LIN {X 0,Y 512.097,Z 685.03,A -85,B 0,C 180,E1 4897.992,E2 4897.992} C_VEL
LIN {X 0,Y 512.114,Z 685.03,A -85,B 0,C 180,E1 4902.666,E2 4902.666} C_VEL
LIN {X 0,Y 512.18,Z 685.03,A -85,B 0,C 180,E1 4907.439,E2 4907.439} C_VEL
LIN {X 0,Y 512.504,Z 685.03,A -85,B 0,C 180,E1 4913.923,E2 4913.923} C_VEL
LIN {X 0,Y 527.673,Z 717.271,A -85,B 0,C 180,E1 4915.573,E2 4915.573} C_VEL
LIN {X 0,Y 526.848,Z 777.404,A -85,B 0,C 180,E1 4916.651,E2 4916.651} C_VEL
LIN {X 0,Y 525.113,Z 815.762,A -85,B 0,C 180,E1 4917.972,E2 4917.972} C_VEL
LIN {X 0,Y 522.678,Z 854.116,A -85,B 0,C 180,E1 4920.009,E2 4920.009} C_VEL
LIN {X 0,Y 520.002,Z 889.911,A -85,B 0,C 180,E1 4922.686,E2 4922.686} C_VEL
LIN {X 0,Y 517.704,Z 920.346,A -85,B 0,C 180,E1 4925.724,E2 4925.724} C_VEL
LIN {X 0,Y 515.761,Z 947.251,A -85,B 0,C 180,E1 4929.222,E2 4929.222} C_VEL
LIN {X 0,Y 514.265,Z 970.27,A -85,B 0,C 180,E1 4933.156,E2 4933.156} C_VEL
LIN {X 0,Y 513.451,Z 987.984,A -85,B 0,C 180,E1 4937.266,E2 4937.266} C_VEL
LIN {X 0,Y 513.157,Z 1000.678,A -85,B 0,C 180,E1 4941.545,E2 4941.545} C_VEL
LIN {X 0,Y 512.98,Z 1006.957,A -85,B 0,C 180,E1 4944.937,E2 4944.937} C_VEL
LIN {X 0,Y 513,Z 1010.088,A -85,B 0,C 180,E1 4948.314,E2 4948.314} C_VEL
LIN {X 0,Y 513.108,Z 1010.088,A -85,B 0,C 180,E1 4951.685,E2 4951.685} C_VEL
LIN {X 0,Y 513.105,Z 1005.755,A -85,B 0,C 180,E1 4955.908,E2 4955.908} C_VEL
LIN {X 0,Y 513.209,Z 996.305,A -85,B 0,C 180,E1 4960.161,E2 4960.161} C_VEL
LIN {X 0,Y 513.736,Z 982.178,A -85,B 0,C 180,E1 4964.236,E2 4964.236} C_VEL
LIN {X 0,Y 514.8,Z 962.363,A -85,B 0,C 180,E1 4968.326,E2 4968.326} C_VEL
LIN {X 0,Y 516.536,Z 936.319,A -85,B 0,C 180,E1 4972.32,E2 4972.32} C_VEL
LIN {X 0,Y 518.821,Z 905.459,A -85,B 0,C 180,E1 4975.866,E2 4975.866} C_VEL
LIN {X 0,Y 521.366,Z 871.94,A -85,B 0,C 180,E1 4978.762,E2 4978.762} C_VEL
LIN {X 0,Y 523.841,Z 836.554,A -85,B 0,C 180,E1 4981.017,E2 4981.017} C_VEL
LIN {X 0,Y 525.931,Z 799.056,A -85,B 0,C 180,E1 4982.681,E2 4982.681} C_VEL
LIN {X 0,Y 527.45,Z 761.276,A -85,B 0,C 180,E1 4983.702,E2 4983.702} C_VEL
LIN {X 0,Y 527.348,Z 716.349,A -85,B 0,C 180,E1 4984.466,E2 4984.466} C_VEL
LIN {X 0,Y 512.508,Z 685.03,A -85,B 0,C 180,E1 4986.077,E2 4986.077} C_VEL
LIN {X 0,Y 512.162,Z 685.03,A -85,B 0,C 180,E1 4992.66,E2 4992.66} C_VEL
LIN {X 0,Y 512.266,Z 685.03,A -85,B 0,C 180,E1 4999.604,E2 4999.604} C_VEL
LIN {X 0,Y 512.378,Z 685.03,A -85,B 0,C 180,E1 5005.55,E2 5005.55} C_VEL
LIN {X 0,Y 512.303,Z 685.03,A -85,B 0,C 180,E1 5009.95,E2 5009.95} C_VEL
LIN {X 0,Y 512.329,Z 685.03,A -85,B 0,C 180,E1 5015.932,E2 5015.932} C_VEL
LIN {X 0,Y 512.467,Z 685.03,A -85,B 0,C 180,E1 5021.099,E2 5021.099} C_VEL
LIN {X 0,Y 512.624,Z 685.03,A -85,B 0,C 180,E1 5026.377,E2 5026.377} C_VEL
LIN {X 0,Y 512.65,Z 685.03,A -85,B 0,C 180,E1 5031.534,E2 5031.534} C_VEL
LIN {X 0,Y 512.92,Z 685.03,A -85,B 0,C 180,E1 5036.624,E2 5036.624} C_VEL
LIN {X 0,Y 513.012,Z 685.03,A -85,B 0,C 180,E1 5041.682,E2 5041.682} C_VEL
LIN {X 0,Y 512.789,Z 685.03,A -85,B 0,C 180,E1 5046.756,E2 5046.756} C_VEL
LIN {X 0,Y 512.606,Z 685.03,A -85,B 0,C 180,E1 5051.888,E2 5051.888} C_VEL
LIN {X 0,Y 512.525,Z 685.03,A -85,B 0,C 180,E1 5057.118,E2 5057.118} C_VEL
LIN {X 0,Y 512.414,Z 685.03,A -85,B 0,C 180,E1 5062.504,E2 5062.504} C_VEL
LIN {X 0,Y 512.263,Z 685.03,A -85,B 0,C 180,E1 5068.114,E2 5068.114} C_VEL
LIN {X 0,Y 512.159,Z 685.03,A -85,B 0,C 180,E1 5074.414,E2 5074.414} C_VEL
LIN {X 0,Y 512.28,Z 685.03,A -85,B 0,C 180,E1 5080.386,E2 5080.386} C_VEL
LIN {X 0,Y 512.179,Z 685.03,A -85,B 0,C 180,E1 5085.001,E2 5085.001} C_VEL
LIN {X 0,Y 512.172,Z 685.03,A -85,B 0,C 180,E1 5091.778,E2 5091.778} C_VEL
LIN {X 0,Y 512.431,Z 685.03,A -85,B 0,C 180,E1 5097.991,E2 5097.991} C_VEL
LIN {X 0,Y 512.52,Z 685.291,A -85,B 0,C 180,E1 5101.148,E2 5101.148} C_VEL
LIN {X 0,Y 521.072,Z 714.374,A -85,B 0,C 180,E1 5103.391,E2 5103.391} C_VEL
LIN {X 0,Y 518.767,Z 750.096,A -85,B 0,C 180,E1 5105.855,E2 5105.855} C_VEL
LIN {X 0,Y 516.704,Z 780.667,A -85,B 0,C 180,E1 5108.764,E2 5108.764} C_VEL
LIN {X 0,Y 515.025,Z 806.913,A -85,B 0,C 180,E1 5112.149,E2 5112.149} C_VEL
LIN {X 0,Y 513.952,Z 827.068,A -85,B 0,C 180,E1 5115.644,E2 5115.644} C_VEL
LIN {X 0,Y 513.394,Z 843.521,A -85,B 0,C 180,E1 5119.617,E2 5119.617} C_VEL
LIN {X 0,Y 513.147,Z 853.42,A -85,B 0,C 180,E1 5123.245,E2 5123.245} C_VEL
LIN {X 0,Y 513.102,Z 858.723,A -85,B 0,C 180,E1 5126.628,E2 5126.628} C_VEL
LIN {X 0,Y 513.002,Z 860.423,A -85,B 0,C 180,E1 5130.379,E2 5130.379} C_VEL
LIN {X 0,Y 513.086,Z 857.628,A -85,B 0,C 180,E1 5134.216,E2 5134.216} C_VEL
LIN {X 0,Y 513.282,Z 849.065,A -85,B 0,C 180,E1 5138.453,E2 5138.453} C_VEL
LIN {X 0,Y 513.64,Z 835.976,A -85,B 0,C 180,E1 5142.298,E2 5142.298} C_VEL
LIN {X 0,Y 514.466,Z 816.847,A -85,B 0,C 180,E1 5146.179,E2 5146.179} C_VEL
LIN {X 0,Y 515.912,Z 793.18,A -85,B 0,C 180,E1 5149.655,E2 5149.655} C_VEL
LIN {X 0,Y 517.757,Z 765.125,A -85,B 0,C 180,E1 5152.734,E2 5152.734} C_VEL
LIN {X 0,Y 519.902,Z 732.834,A -85,B 0,C 180,E1 5155.348,E2 5155.348} C_VEL
LIN {X 0,Y 520.429,Z 711.081,A -85,B 0,C 180,E1 5156.776,E2 5156.776} C_VEL
LIN {X 0,Y 513.339,Z 688.629,A -85,B 0,C 180,E1 5158.542,E2 5158.542} C_VEL
LIN {X 0,Y 512.428,Z 685.03,A -85,B 0,C 180,E1 5158.781,E2 5158.781} C_VEL
LIN {X 0,Y 512.245,Z 685.03,A -85,B 0,C 180,E1 5164.44,E2 5164.44} C_VEL
LIN {X 0,Y 512.172,Z 685.03,A -85,B 0,C 180,E1 5170.404,E2 5170.404} C_VEL
LIN {X 0,Y 512.18,Z 685.03,A -85,B 0,C 180,E1 5175.01,E2 5175.01} C_VEL
LIN {X 0,Y 512.298,Z 685.03,A -85,B 0,C 180,E1 5179.982,E2 5179.982} C_VEL
LIN {X 0,Y 512.199,Z 685.03,A -85,B 0,C 180,E1 5185.968,E2 5185.968} C_VEL
LIN {X 0,Y 512.303,Z 685.03,A -85,B 0,C 180,E1 5192.086,E2 5192.086} C_VEL
LIN {X 0,Y 512.422,Z 685.03,A -85,B 0,C 180,E1 5197.496,E2 5197.496} C_VEL
LIN {X 0,Y 512.61,Z 685.03,A -85,B 0,C 180,E1 5202.885,E2 5202.885} C_VEL
LIN {X 0,Y 512.652,Z 685.03,A -85,B 0,C 180,E1 5208.113,E2 5208.113} C_VEL
LIN {X 0,Y 512.68,Z 685.03,A -85,B 0,C 180,E1 5213.242,E2 5213.242} C_VEL
LIN {X 0,Y 512.709,Z 685.03,A -85,B 0,C 180,E1 5218.317,E2 5218.317} C_VEL
LIN {X 0,Y 512.758,Z 685.03,A -85,B 0,C 180,E1 5223.377,E2 5223.377} C_VEL
LIN {X 0,Y 512.593,Z 685.03,A -85,B 0,C 180,E1 5228.467,E2 5228.467} C_VEL
LIN {X 0,Y 512.526,Z 685.03,A -85,B 0,C 180,E1 5233.689,E2 5233.689} C_VEL
LIN {X 0,Y 512.406,Z 685.03,A -85,B 0,C 180,E1 5239.546,E2 5239.546} C_VEL
LIN {X 0,Y 512.335,Z 685.03,A -85,B 0,C 180,E1 5244.354,E2 5244.354} C_VEL
LIN {X 0,Y 512.197,Z 685.03,A -85,B 0,C 180,E1 5250.057,E2 5250.057} C_VEL
LIN {X 0,Y 512.084,Z 685.03,A -85,B 0,C 180,E1 5256.112,E2 5256.112} C_VEL
LIN {X 0,Y 512.097,Z 685.03,A -85,B 0,C 180,E1 5257.992,E2 5257.992} C_VEL
LIN {X 0,Y 509.625,Z 685.03,A -85,B 0,C 180,E1 5259.422,E2 5259.422} C_VEL
LIN {X 0,Y 504.094,Z 685.03,A -85,B 0,C 180,E1 5261.814,E2 5261.814} C_VEL
LIN {X 0,Y 504.227,Z 685.03,A -85,B 0,C 180,E1 5268.432,E2 5268.432} C_VEL
LIN {X 0,Y 504.534,Z 685.03,A -85,B 0,C 180,E1 5273.399,E2 5273.399} C_VEL
LIN {X 0,Y 515.554,Z 708.405,A -85,B 0,C 180,E1 5274.539,E2 5274.539} C_VEL
LIN {X 0,Y 521.274,Z 720.033,A -85,B 0,C 180,E1 5275.135,E2 5275.135} C_VEL
LIN {X 0,Y 520.263,Z 777.402,A -85,B 0,C 180,E1 5276.172,E2 5276.172} C_VEL
LIN {X 0,Y 518.336,Z 816.284,A -85,B 0,C 180,E1 5277.529,E2 5277.529} C_VEL
LIN {X 0,Y 515.69,Z 854.113,A -85,B 0,C 180,E1 5279.56,E2 5279.56} C_VEL
LIN {X 0,Y 512.844,Z 889.613,A -85,B 0,C 180,E1 5282.245,E2 5282.245} C_VEL
LIN {X 0,Y 510.294,Z 920.539,A -85,B 0,C 180,E1 5285.372,E2 5285.372} C_VEL
LIN {X 0,Y 508.137,Z 947.251,A -85,B 0,C 180,E1 5288.895,E2 5288.895} C_VEL
LIN {X 0,Y 506.553,Z 970.269,A -85,B 0,C 180,E1 5292.892,E2 5292.892} C_VEL
LIN {X 0,Y 505.631,Z 987.985,A -85,B 0,C 180,E1 5297.066,E2 5297.066} C_VEL
LIN {X 0,Y 505.264,Z 1000.678,A -85,B 0,C 180,E1 5301.412,E2 5301.412} C_VEL
LIN {X 0,Y 505.087,Z 1006.957,A -85,B 0,C 180,E1 5304.858,E2 5304.858} C_VEL
LIN {X 0,Y 505.097,Z 1010.088,A -85,B 0,C 180,E1 5308.288,E2 5308.288} C_VEL
LIN {X 0,Y 505.201,Z 1010.089,A -85,B 0,C 180,E1 5311.712,E2 5311.712} C_VEL
LIN {X 0,Y 505.213,Z 1005.755,A -85,B 0,C 180,E1 5316.001,E2 5316.001} C_VEL
LIN {X 0,Y 505.327,Z 996.305,A -85,B 0,C 180,E1 5320.321,E2 5320.321} C_VEL
LIN {X 0,Y 505.99,Z 981.084,A -85,B 0,C 180,E1 5324.736,E2 5324.736} C_VEL
LIN {X 0,Y 507.259,Z 959.66,A -85,B 0,C 180,E1 5329.101,E2 5329.101} C_VEL
LIN {X 0,Y 509.092,Z 934.49,A -85,B 0,C 180,E1 5332.91,E2 5332.91} C_VEL
LIN {X 0,Y 511.629,Z 904.316,A -85,B 0,C 180,E1 5336.375,E2 5336.375} C_VEL
LIN {X 0,Y 514.424,Z 870.414,A -85,B 0,C 180,E1 5339.307,E2 5339.307} C_VEL
LIN {X 0,Y 517.101,Z 834.197,A -85,B 0,C 180,E1 5341.602,E2 5341.602} C_VEL
LIN {X 0,Y 519.376,Z 795.774,A -85,B 0,C 180,E1 5343.27,E2 5343.27} C_VEL
LIN {X 0,Y 520.962,Z 758.124,A -85,B 0,C 180,E1 5344.241,E2 5344.241} C_VEL
LIN {X 0,Y 520.802,Z 718.82,A -85,B 0,C 180,E1 5344.922,E2 5344.922} C_VEL
LIN {X 0,Y 504.596,Z 686.097,A -85,B 0,C 180,E1 5346.569,E2 5346.569} C_VEL
LIN {X 0,Y 504.518,Z 685.03,A -85,B 0,C 180,E1 5346.74,E2 5346.74} C_VEL
LIN {X 0,Y 504.156,Z 685.03,A -85,B 0,C 180,E1 5353.505,E2 5353.505} C_VEL
LIN {X 0,Y 504.253,Z 685.03,A -85,B 0,C 180,E1 5358.825,E2 5358.825} C_VEL
LIN {X 0,Y 504.465,Z 685.03,A -85,B 0,C 180,E1 5365.364,E2 5365.364} C_VEL
LIN {X 0,Y 504.332,Z 685.03,A -85,B 0,C 180,E1 5371.396,E2 5371.396} C_VEL
LIN {X 0,Y 504.369,Z 685.03,A -85,B 0,C 180,E1 5377.11,E2 5377.11} C_VEL
LIN {X 0,Y 504.613,Z 685.03,A -85,B 0,C 180,E1 5383.122,E2 5383.122} C_VEL
LIN {X 0,Y 504.654,Z 685.03,A -85,B 0,C 180,E1 5387.916,E2 5387.916} C_VEL
LIN {X 0,Y 504.756,Z 685.03,A -85,B 0,C 180,E1 5393.129,E2 5393.129} C_VEL
LIN {X 0,Y 504.835,Z 685.03,A -85,B 0,C 180,E1 5398.284,E2 5398.284} C_VEL
LIN {X 0,Y 504.85,Z 685.03,A -85,B 0,C 180,E1 5403.424,E2 5403.424} C_VEL
LIN {X 0,Y 504.668,Z 685.03,A -85,B 0,C 180,E1 5409.347,E2 5409.347} C_VEL
LIN {X 0,Y 504.586,Z 685.03,A -85,B 0,C 180,E1 5415.609,E2 5415.609} C_VEL
LIN {X 0,Y 504.482,Z 685.03,A -85,B 0,C 180,E1 5421.988,E2 5421.988} C_VEL
LIN {X 0,Y 504.387,Z 685.03,A -85,B 0,C 180,E1 5426.658,E2 5426.658} C_VEL
LIN {X 0,Y 504.208,Z 685.03,A -85,B 0,C 180,E1 5433.072,E2 5433.072} C_VEL
LIN {X 0,Y 504.345,Z 685.03,A -85,B 0,C 180,E1 5438.93,E2 5438.93} C_VEL
LIN {X 0,Y 504.223,Z 685.03,A -85,B 0,C 180,E1 5444.09,E2 5444.09} C_VEL
LIN {X 0,Y 504.155,Z 685.03,A -85,B 0,C 180,E1 5448.816,E2 5448.816} C_VEL
LIN {X 0,Y 504.344,Z 685.03,A -85,B 0,C 180,E1 5455.356,E2 5455.356} C_VEL
LIN {X 0,Y 504.555,Z 685.116,A -85,B 0,C 180,E1 5460.483,E2 5460.483} C_VEL
LIN {X 0,Y 513.153,Z 711.842,A -85,B 0,C 180,E1 5462.61,E2 5462.61} C_VEL
LIN {X 0,Y 514.053,Z 720.156,A -85,B 0,C 180,E1 5463.228,E2 5463.228} C_VEL
LIN {X 0,Y 511.446,Z 752.039,A -85,B 0,C 180,E1 5465.603,E2 5465.603} C_VEL
LIN {X 0,Y 508.858,Z 784.682,A -85,B 0,C 180,E1 5468.9,E2 5468.9} C_VEL
LIN {X 0,Y 507.106,Z 810.967,A -85,B 0,C 180,E1 5472.498,E2 5472.498} C_VEL
LIN {X 0,Y 506.093,Z 830.729,A -85,B 0,C 180,E1 5476.2,E2 5476.2} C_VEL
LIN {X 0,Y 505.493,Z 845.971,A -85,B 0,C 180,E1 5480.244,E2 5480.244} C_VEL
LIN {X 0,Y 505.249,Z 855.071,A -85,B 0,C 180,E1 5484,E2 5484} C_VEL
LIN {X 0,Y 505.149,Z 860.041,A -85,B 0,C 180,E1 5488.288,E2 5488.288} C_VEL
LIN {X 0,Y 505.186,Z 859.987,A -85,B 0,C 180,E1 5491.712,E2 5491.712} C_VEL
LIN {X 0,Y 505.182,Z 854.908,A -85,B 0,C 180,E1 5496.001,E2 5496.001} C_VEL
LIN {X 0,Y 505.454,Z 845.208,A -85,B 0,C 180,E1 5499.917,E2 5499.917} C_VEL
LIN {X 0,Y 506.05,Z 830.338,A -85,B 0,C 180,E1 5503.801,E2 5503.801} C_VEL
LIN {X 0,Y 507.204,Z 809.134,A -85,B 0,C 180,E1 5507.702,E2 5507.702} C_VEL
LIN {X 0,Y 508.952,Z 783.691,A -85,B 0,C 180,E1 5511.124,E2 5511.124} C_VEL
LIN {X 0,Y 511.502,Z 751.027,A -85,B 0,C 180,E1 5514.394,E2 5514.394} C_VEL
LIN {X 0,Y 514.064,Z 719.213,A -85,B 0,C 180,E1 5516.745,E2 5516.745} C_VEL
LIN {X 0,Y 510.499,Z 701.311,A -85,B 0,C 180,E1 5518.129,E2 5518.129} C_VEL
LIN {X 0,Y 504.49,Z 685.03,A -85,B 0,C 180,E1 5519.468,E2 5519.468} C_VEL
LIN {X 0,Y 504.325,Z 685.03,A -85,B 0,C 180,E1 5524.646,E2 5524.646} C_VEL
LIN {X 0,Y 504.176,Z 685.03,A -85,B 0,C 180,E1 5531.182,E2 5531.182} C_VEL
LIN {X 0,Y 504.21,Z 685.03,A -85,B 0,C 180,E1 5536.51,E2 5536.51} C_VEL
LIN {X 0,Y 504.346,Z 685.03,A -85,B 0,C 180,E1 5541.082,E2 5541.082} C_VEL
LIN {X 0,Y 504.258,Z 685.03,A -85,B 0,C 180,E1 5546.919,E2 5546.919} C_VEL
LIN {X 0,Y 504.401,Z 685.03,A -85,B 0,C 180,E1 5553.342,E2 5553.342} C_VEL
LIN {X 0,Y 504.566,Z 685.03,A -85,B 0,C 180,E1 5558.974,E2 5558.974} C_VEL
LIN {X 0,Y 504.723,Z 685.03,A -85,B 0,C 180,E1 5564.395,E2 5564.395} C_VEL
LIN {X 0,Y 504.738,Z 685.03,A -85,B 0,C 180,E1 5570.605,E2 5570.605} C_VEL
LIN {X 0,Y 504.949,Z 685.03,A -85,B 0,C 180,E1 5576.577,E2 5576.577} C_VEL
LIN {X 0,Y 505.107,Z 685.03,A -85,B 0,C 180,E1 5581.715,E2 5581.715} C_VEL
LIN {X 0,Y 504.854,Z 685.03,A -85,B 0,C 180,E1 5586.869,E2 5586.869} C_VEL
LIN {X 0,Y 504.672,Z 685.03,A -85,B 0,C 180,E1 5592.084,E2 5592.084} C_VEL
LIN {X 0,Y 504.596,Z 685.03,A -85,B 0,C 180,E1 5597.403,E2 5597.403} C_VEL
LIN {X 0,Y 504.42,Z 685.03,A -85,B 0,C 180,E1 5602.888,E2 5602.888} C_VEL
LIN {X 0,Y 504.299,Z 685.03,A -85,B 0,C 180,E1 5608.606,E2 5608.606} C_VEL
LIN {X 0,Y 504.178,Z 685.03,A -85,B 0,C 180,E1 5614.658,E2 5614.658} C_VEL
LIN {X 0,Y 504.135,Z 685.03,A -85,B 0,C 180,E1 5621.187,E2 5621.187} C_VEL
LIN {X 0,Y 504.094,Z 685.03,A -85,B 0,C 180,E1 5621.814,E2 5621.814} C_VEL
LIN {X 0,Y 500.142,Z 685.03,A -85,B 0,C 180,E1 5623.763,E2 5623.763} C_VEL
LIN {X 0,Y 496.227,Z 685.03,A -85,B 0,C 180,E1 5625.743,E2 5625.743} C_VEL
LIN {X 0,Y 496.487,Z 685.03,A -85,B 0,C 180,E1 5632.207,E2 5632.207} C_VEL
LIN {X 0,Y 496.53,Z 685.03,A -85,B 0,C 180,E1 5632.806,E2 5632.806} C_VEL
LIN {X 0,Y 514.548,Z 722.423,A -85,B 0,C 180,E1 5634.696,E2 5634.696} C_VEL
LIN {X 0,Y 513.689,Z 777.228,A -85,B 0,C 180,E1 5635.675,E2 5635.675} C_VEL
LIN {X 0,Y 511.692,Z 815.212,A -85,B 0,C 180,E1 5637,E2 5637} C_VEL
LIN {X 0,Y 508.795,Z 853.576,A -85,B 0,C 180,E1 5639.064,E2 5639.064} C_VEL
LIN {X 0,Y 505.71,Z 889.194,A -85,B 0,C 180,E1 5641.778,E2 5641.778} C_VEL
LIN {X 0,Y 502.9,Z 920.736,A -85,B 0,C 180,E1 5645.01,E2 5645.01} C_VEL
LIN {X 0,Y 500.43,Z 948.703,A -85,B 0,C 180,E1 5648.786,E2 5648.786} C_VEL
LIN {X 0,Y 498.726,Z 971.348,A -85,B 0,C 180,E1 5652.842,E2 5652.842} C_VEL
LIN {X 0,Y 497.8,Z 987.985,A -85,B 0,C 180,E1 5656.859,E2 5656.859} C_VEL
LIN {X 0,Y 497.389,Z 1000.678,A -85,B 0,C 180,E1 5661.275,E2 5661.275} C_VEL
LIN {X 0,Y 497.195,Z 1006.958,A -85,B 0,C 180,E1 5664.776,E2 5664.776} C_VEL
LIN {X 0,Y 497.219,Z 1010.088,A -85,B 0,C 180,E1 5668.261,E2 5668.261} C_VEL
LIN {X 0,Y 497.297,Z 1010.089,A -85,B 0,C 180,E1 5671.739,E2 5671.739} C_VEL
LIN {X 0,Y 497.335,Z 1005.755,A -85,B 0,C 180,E1 5676.096,E2 5676.096} C_VEL
LIN {X 0,Y 497.446,Z 996.305,A -85,B 0,C 180,E1 5680.487,E2 5680.487} C_VEL
LIN {X 0,Y 498.25,Z 980.677,A -85,B 0,C 180,E1 5685.075,E2 5685.075} C_VEL
LIN {X 0,Y 499.593,Z 959.659,A -85,B 0,C 180,E1 5689.405,E2 5689.405} C_VEL
LIN {X 0,Y 501.627,Z 934.489,A -85,B 0,C 180,E1 5693.271,E2 5693.271} C_VEL
LIN {X 0,Y 504.34,Z 904.418,A -85,B 0,C 180,E1 5696.776,E2 5696.776} C_VEL
LIN {X 0,Y 507.375,Z 870.403,A -85,B 0,C 180,E1 5699.756,E2 5699.756} C_VEL
LIN {X 0,Y 510.324,Z 833.875,A -85,B 0,C 180,E1 5702.09,E2 5702.09} C_VEL
LIN {X 0,Y 512.737,Z 795.659,A -85,B 0,C 180,E1 5703.763,E2 5703.763} C_VEL
LIN {X 0,Y 514.364,Z 760.078,A -85,B 0,C 180,E1 5704.694,E2 5704.694} C_VEL
LIN {X 0,Y 513.905,Z 720.91,A -85,B 0,C 180,E1 5705.369,E2 5705.369} C_VEL
LIN {X 0,Y 496.532,Z 685.03,A -85,B 0,C 180,E1 5707.193,E2 5707.193} C_VEL
LIN {X 0,Y 496.25,Z 685.03,A -85,B 0,C 180,E1 5713.131,E2 5713.131} C_VEL
LIN {X 0,Y 496.321,Z 685.03,A -85,B 0,C 180,E1 5719.472,E2 5719.472} C_VEL
LIN {X 0,Y 496.56,Z 685.03,A -85,B 0,C 180,E1 5725.135,E2 5725.135} C_VEL
LIN {X 0,Y 496.442,Z 685.03,A -85,B 0,C 180,E1 5730.898,E2 5730.898} C_VEL
LIN {X 0,Y 496.419,Z 685.03,A -85,B 0,C 180,E1 5736.722,E2 5736.722} C_VEL
LIN {X 0,Y 496.68,Z 685.03,A -85,B 0,C 180,E1 5742.311,E2 5742.311} C_VEL
LIN {X 0,Y 496.738,Z 685.03,A -85,B 0,C 180,E1 5747.72,E2 5747.72} C_VEL
LIN {X 0,Y 496.871,Z 685.03,A -85,B 0,C 180,E1 5753.02,E2 5753.02} C_VEL
LIN {X 0,Y 496.958,Z 685.03,A -85,B 0,C 180,E1 5758.257,E2 5758.257} C_VEL
LIN {X 0,Y 496.965,Z 685.03,A -85,B 0,C 180,E1 5763.478,E2 5763.478} C_VEL
LIN {X 0,Y 496.787,Z 685.03,A -85,B 0,C 180,E1 5768.732,E2 5768.732} C_VEL
LIN {X 0,Y 496.754,Z 685.03,A -85,B 0,C 180,E1 5774.06,E2 5774.06} C_VEL
LIN {X 0,Y 496.61,Z 685.03,A -85,B 0,C 180,E1 5779.616,E2 5779.616} C_VEL
LIN {X 0,Y 496.494,Z 685.03,A -85,B 0,C 180,E1 5785.177,E2 5785.177} C_VEL
LIN {X 0,Y 496.265,Z 685.03,A -85,B 0,C 180,E1 5791.636,E2 5791.636} C_VEL
LIN {X 0,Y 496.382,Z 685.03,A -85,B 0,C 180,E1 5797.778,E2 5797.778} C_VEL
LIN {X 0,Y 496.305,Z 685.03,A -85,B 0,C 180,E1 5804.362,E2 5804.362} C_VEL
LIN {X 0,Y 496.213,Z 685.03,A -85,B 0,C 180,E1 5810.312,E2 5810.312} C_VEL
LIN {X 0,Y 496.479,Z 685.03,A -85,B 0,C 180,E1 5816.832,E2 5816.832} C_VEL
LIN {X 0,Y 496.665,Z 685.438,A -85,B 0,C 180,E1 5819.81,E2 5819.81} C_VEL
LIN {X 0,Y 505.807,Z 711.87,A -85,B 0,C 180,E1 5822.019,E2 5822.019} C_VEL
LIN {X 0,Y 507.328,Z 721.922,A -85,B 0,C 180,E1 5822.81,E2 5822.81} C_VEL
LIN {X 0,Y 504.5,Z 754.004,A -85,B 0,C 180,E1 5825.244,E2 5825.244} C_VEL
LIN {X 0,Y 501.775,Z 781.617,A -85,B 0,C 180,E1 5828.151,E2 5828.151} C_VEL
LIN {X 0,Y 499.435,Z 810.492,A -85,B 0,C 180,E1 5832.139,E2 5832.139} C_VEL
LIN {X 0,Y 498.271,Z 830.725,A -85,B 0,C 180,E1 5835.979,E2 5835.979} C_VEL
LIN {X 0,Y 497.603,Z 845.969,A -85,B 0,C 180,E1 5840.087,E2 5840.087} C_VEL
LIN {X 0,Y 497.368,Z 855.069,A -85,B 0,C 180,E1 5843.904,E2 5843.904} C_VEL
LIN {X 0,Y 497.247,Z 860.04,A -85,B 0,C 180,E1 5848.261,E2 5848.261} C_VEL
LIN {X 0,Y 497.306,Z 859.987,A -85,B 0,C 180,E1 5851.739,E2 5851.739} C_VEL
LIN {X 0,Y 497.309,Z 854.909,A -85,B 0,C 180,E1 5856.096,E2 5856.096} C_VEL
LIN {X 0,Y 497.564,Z 845.802,A -85,B 0,C 180,E1 5859.879,E2 5859.879} C_VEL
LIN {X 0,Y 498.244,Z 830.341,A -85,B 0,C 180,E1 5864.022,E2 5864.022} C_VEL
LIN {X 0,Y 499.476,Z 809.884,A -85,B 0,C 180,E1 5867.868,E2 5867.868} C_VEL
LIN {X 0,Y 501.832,Z 780.942,A -85,B 0,C 180,E1 5871.846,E2 5871.846} C_VEL
LIN {X 0,Y 504.673,Z 751.737,A -85,B 0,C 180,E1 5874.864,E2 5874.864} C_VEL
LIN {X 0,Y 507.472,Z 719.393,A -85,B 0,C 180,E1 5877.262,E2 5877.262} C_VEL
LIN {X 0,Y 501.872,Z 698.659,A -85,B 0,C 180,E1 5878.986,E2 5878.986} C_VEL
LIN {X 0,Y 496.536,Z 685.03,A -85,B 0,C 180,E1 5880.178,E2 5880.178} C_VEL
LIN {X 0,Y 496.376,Z 685.03,A -85,B 0,C 180,E1 5885.282,E2 5885.282} C_VEL
LIN {X 0,Y 496.223,Z 685.03,A -85,B 0,C 180,E1 5891.991,E2 5891.991} C_VEL
LIN {X 0,Y 496.312,Z 685.03,A -85,B 0,C 180,E1 5898.027,E2 5898.027} C_VEL
LIN {X 0,Y 496.383,Z 685.03,A -85,B 0,C 180,E1 5902.563,E2 5902.563} C_VEL
LIN {X 0,Y 496.344,Z 685.03,A -85,B 0,C 180,E1 5908.886,E2 5908.886} C_VEL
LIN {X 0,Y 496.503,Z 685.03,A -85,B 0,C 180,E1 5914.824,E2 5914.824} C_VEL
LIN {X 0,Y 496.67,Z 685.03,A -85,B 0,C 180,E1 5920.481,E2 5920.481} C_VEL
LIN {X 0,Y 496.932,Z 685.03,A -85,B 0,C 180,E1 5926.341,E2 5926.341} C_VEL
LIN {X 0,Y 496.884,Z 685.03,A -85,B 0,C 180,E1 5933.027,E2 5933.027} C_VEL
LIN {X 0,Y 496.935,Z 685.03,A -85,B 0,C 180,E1 5938.263,E2 5938.263} C_VEL
LIN {X 0,Y 496.968,Z 685.03,A -85,B 0,C 180,E1 5943.485,E2 5943.485} C_VEL
LIN {X 0,Y 496.787,Z 685.03,A -85,B 0,C 180,E1 5948.738,E2 5948.738} C_VEL
LIN {X 0,Y 496.695,Z 685.03,A -85,B 0,C 180,E1 5954.069,E2 5954.069} C_VEL
LIN {X 0,Y 496.589,Z 685.03,A -85,B 0,C 180,E1 5959.61,E2 5959.61} C_VEL
LIN {X 0,Y 496.483,Z 685.03,A -85,B 0,C 180,E1 5965.185,E2 5965.185} C_VEL
LIN {X 0,Y 496.261,Z 685.03,A -85,B 0,C 180,E1 5971.636,E2 5971.636} C_VEL
LIN {X 0,Y 496.185,Z 685.03,A -85,B 0,C 180,E1 5977.748,E2 5977.748} C_VEL
LIN {X 0,Y 496.221,Z 685.03,A -85,B 0,C 180,E1 5984.381,E2 5984.381} C_VEL
LIN {X 0,Y 496.227,Z 685.03,A -85,B 0,C 180,E1 5985.743,E2 5985.743} C_VEL
LIN {X 0,Y 492.303,Z 685.03,A -85,B 0,C 180,E1 5987.718,E2 5987.718} C_VEL
LIN {X 0,Y 488.416,Z 685.03,A -85,B 0,C 180,E1 5989.726,E2 5989.726} C_VEL
LIN {X 0,Y 488.646,Z 685.828,A -85,B 0,C 180,E1 5992.272,E2 5992.272} C_VEL
LIN {X 0,Y 507.762,Z 724.889,A -85,B 0,C 180,E1 5994.287,E2 5994.287} C_VEL
LIN {X 0,Y 506.719,Z 778.267,A -85,B 0,C 180,E1 5995.271,E2 5995.271} C_VEL
LIN {X 0,Y 504.74,Z 817.548,A -85,B 0,C 180,E1 5996.637,E2 5996.637} C_VEL
LIN {X 0,Y 501.902,Z 853.739,A -85,B 0,C 180,E1 5998.603,E2 5998.603} C_VEL
LIN {X 0,Y 498.582,Z 889.477,A -85,B 0,C 180,E1 6001.366,E2 6001.366} C_VEL
LIN {X 0,Y 495.511,Z 920.932,A -85,B 0,C 180,E1 6004.636,E2 6004.636} C_VEL
LIN {X 0,Y 492.868,Z 948.701,A -85,B 0,C 180,E1 6008.445,E2 6008.445} C_VEL
LIN {X 0,Y 491.139,Z 969.896,A -85,B 0,C 180,E1 6012.259,E2 6012.259} C_VEL
LIN {X 0,Y 490.003,Z 987.984,A -85,B 0,C 180,E1 6016.646,E2 6016.646} C_VEL
LIN {X 0,Y 489.507,Z 1000.678,A -85,B 0,C 180,E1 6021.133,E2 6021.133} C_VEL
LIN {X 0,Y 489.305,Z 1006.957,A -85,B 0,C 180,E1 6024.691,E2 6024.691} C_VEL
LIN {X 0,Y 489.316,Z 1010.088,A -85,B 0,C 180,E1 6028.233,E2 6028.233} C_VEL
LIN {X 0,Y 489.39,Z 1010.089,A -85,B 0,C 180,E1 6031.767,E2 6031.767} C_VEL
LIN {X 0,Y 489.44,Z 1005.755,A -85,B 0,C 180,E1 6036.195,E2 6036.195} C_VEL
LIN {X 0,Y 489.582,Z 996.305,A -85,B 0,C 180,E1 6040.657,E2 6040.657} C_VEL
LIN {X 0,Y 490.407,Z 981.289,A -85,B 0,C 180,E1 6045.162,E2 6045.162} C_VEL
LIN {X 0,Y 491.944,Z 959.657,A -85,B 0,C 180,E1 6049.719,E2 6049.719} C_VEL
LIN {X 0,Y 494.27,Z 933.457,A -85,B 0,C 180,E1 6053.779,E2 6053.779} C_VEL
LIN {X 0,Y 497.191,Z 903.531,A -85,B 0,C 180,E1 6057.287,E2 6057.287} C_VEL
LIN {X 0,Y 500.402,Z 870.4,A -85,B 0,C 180,E1 6060.213,E2 6060.213} C_VEL
LIN {X 0,Y 503.49,Z 834.853,A -85,B 0,C 180,E1 6062.52,E2 6062.52} C_VEL
LIN {X 0,Y 505.783,Z 797.933,A -85,B 0,C 180,E1 6064.128,E2 6064.128} C_VEL
LIN {X 0,Y 507.55,Z 758.035,A -85,B 0,C 180,E1 6065.17,E2 6065.17} C_VEL
LIN {X 0,Y 507.314,Z 723.989,A -85,B 0,C 180,E1 6065.758,E2 6065.758} C_VEL
LIN {X 0,Y 488.681,Z 686.145,A -85,B 0,C 180,E1 6067.733,E2 6067.733} C_VEL
LIN {X 0,Y 488.582,Z 685.03,A -85,B 0,C 180,E1 6067.82,E2 6067.82} C_VEL
LIN {X 0,Y 488.335,Z 685.03,A -85,B 0,C 180,E1 6074.706,E2 6074.706} C_VEL
LIN {X 0,Y 488.463,Z 685.03,A -85,B 0,C 180,E1 6080.562,E2 6080.562} C_VEL
LIN {X 0,Y 488.604,Z 685.03,A -85,B 0,C 180,E1 6086.497,E2 6086.497} C_VEL
LIN {X 0,Y 488.47,Z 685.03,A -85,B 0,C 180,E1 6092.393,E2 6092.393} C_VEL
LIN {X 0,Y 488.545,Z 685.03,A -85,B 0,C 180,E1 6098.242,E2 6098.242} C_VEL
LIN {X 0,Y 488.773,Z 685.03,A -85,B 0,C 180,E1 6103.865,E2 6103.865} C_VEL
LIN {X 0,Y 488.855,Z 685.03,A -85,B 0,C 180,E1 6109.324,E2 6109.324} C_VEL
LIN {X 0,Y 489.064,Z 685.03,A -85,B 0,C 180,E1 6114.686,E2 6114.686} C_VEL
LIN {X 0,Y 489.155,Z 685.03,A -85,B 0,C 180,E1 6119.997,E2 6119.997} C_VEL
LIN {X 0,Y 489.072,Z 685.03,A -85,B 0,C 180,E1 6125.307,E2 6125.307} C_VEL
LIN {X 0,Y 488.867,Z 685.03,A -85,B 0,C 180,E1 6130.669,E2 6130.669} C_VEL
LIN {X 0,Y 488.719,Z 685.03,A -85,B 0,C 180,E1 6136.83,E2 6136.83} C_VEL
LIN {X 0,Y 488.631,Z 685.03,A -85,B 0,C 180,E1 6142.111,E2 6142.111} C_VEL
LIN {X 0,Y 488.477,Z 685.03,A -85,B 0,C 180,E1 6147.599,E2 6147.599} C_VEL
LIN {X 0,Y 488.397,Z 685.03,A -85,B 0,C 180,E1 6153.783,E2 6153.783} C_VEL
LIN {X 0,Y 488.426,Z 685.03,A -85,B 0,C 180,E1 6160.443,E2 6160.443} C_VEL
LIN {X 0,Y 488.373,Z 685.03,A -85,B 0,C 180,E1 6165.28,E2 6165.28} C_VEL
LIN {X 0,Y 488.313,Z 685.03,A -85,B 0,C 180,E1 6171.827,E2 6171.827} C_VEL
LIN {X 0,Y 488.592,Z 685.03,A -85,B 0,C 180,E1 6178.329,E2 6178.329} C_VEL
LIN {X 0,Y 488.725,Z 685.847,A -85,B 0,C 180,E1 6179.113,E2 6179.113} C_VEL
LIN {X 0,Y 498.407,Z 711.719,A -85,B 0,C 180,E1 6181.389,E2 6181.389} C_VEL
LIN {X 0,Y 500.537,Z 724.804,A -85,B 0,C 180,E1 6182.45,E2 6182.45} C_VEL
LIN {X 0,Y 497.572,Z 755.94,A -85,B 0,C 180,E1 6184.876,E2 6184.876} C_VEL
LIN {X 0,Y 494.651,Z 783.367,A -85,B 0,C 180,E1 6187.82,E2 6187.82} C_VEL
LIN {X 0,Y 492.081,Z 807.489,A -85,B 0,C 180,E1 6191.31,E2 6191.31} C_VEL
LIN {X 0,Y 490.436,Z 830.721,A -85,B 0,C 180,E1 6195.75,E2 6195.75} C_VEL
LIN {X 0,Y 489.721,Z 846.054,A -85,B 0,C 180,E1 6199.956,E2 6199.956} C_VEL
LIN {X 0,Y 489.476,Z 855.067,A -85,B 0,C 180,E1 6203.806,E2 6203.806} C_VEL
LIN {X 0,Y 489.345,Z 860.039,A -85,B 0,C 180,E1 6208.233,E2 6208.233} C_VEL
LIN {X 0,Y 489.402,Z 859.987,A -85,B 0,C 180,E1 6211.767,E2 6211.767} C_VEL
LIN {X 0,Y 489.422,Z 854.91,A -85,B 0,C 180,E1 6216.195,E2 6216.195} C_VEL
LIN {X 0,Y 489.691,Z 845.828,A -85,B 0,C 180,E1 6220.031,E2 6220.031} C_VEL
LIN {X 0,Y 490.449,Z 830.343,A -85,B 0,C 180,E1 6224.249,E2 6224.249} C_VEL
LIN {X 0,Y 492.221,Z 806.424,A -85,B 0,C 180,E1 6228.777,E2 6228.777} C_VEL
LIN {X 0,Y 494.868,Z 780.901,A -85,B 0,C 180,E1 6232.406,E2 6232.406} C_VEL
LIN {X 0,Y 497.975,Z 751.495,A -85,B 0,C 180,E1 6235.43,E2 6235.43} C_VEL
LIN {X 0,Y 500.459,Z 720.228,A -85,B 0,C 180,E1 6237.786,E2 6237.786} C_VEL
LIN {X 0,Y 494.253,Z 699.278,A -85,B 0,C 180,E1 6239.622,E2 6239.622} C_VEL
LIN {X 0,Y 488.601,Z 685.03,A -85,B 0,C 180,E1 6240.886,E2 6240.886} C_VEL
LIN {X 0,Y 488.352,Z 685.03,A -85,B 0,C 180,E1 6246.556,E2 6246.556} C_VEL
LIN {X 0,Y 488.323,Z 685.03,A -85,B 0,C 180,E1 6252.831,E2 6252.831} C_VEL
LIN {X 0,Y 488.401,Z 685.03,A -85,B 0,C 180,E1 6257.861,E2 6257.861} C_VEL
LIN {X 0,Y 488.415,Z 685.03,A -85,B 0,C 180,E1 6264.061,E2 6264.061} C_VEL
LIN {X 0,Y 488.428,Z 685.03,A -85,B 0,C 180,E1 6270.381,E2 6270.381} C_VEL
LIN {X 0,Y 488.622,Z 685.03,A -85,B 0,C 180,E1 6276.335,E2 6276.335} C_VEL
LIN {X 0,Y 488.808,Z 685.03,A -85,B 0,C 180,E1 6282.024,E2 6282.024} C_VEL
LIN {X 0,Y 488.956,Z 685.03,A -85,B 0,C 180,E1 6287.528,E2 6287.528} C_VEL
LIN {X 0,Y 488.969,Z 685.03,A -85,B 0,C 180,E1 6292.913,E2 6292.913} C_VEL
LIN {X 0,Y 489.034,Z 685.03,A -85,B 0,C 180,E1 6298.235,E2 6298.235} C_VEL
LIN {X 0,Y 489.062,Z 685.03,A -85,B 0,C 180,E1 6303.541,E2 6303.541} C_VEL
LIN {X 0,Y 488.86,Z 685.03,A -85,B 0,C 180,E1 6308.973,E2 6308.973} C_VEL
LIN {X 0,Y 488.764,Z 685.03,A -85,B 0,C 180,E1 6314.302,E2 6314.302} C_VEL
LIN {X 0,Y 488.676,Z 685.03,A -85,B 0,C 180,E1 6319.859,E2 6319.859} C_VEL
LIN {X 0,Y 488.463,Z 685.03,A -85,B 0,C 180,E1 6326.377,E2 6326.377} C_VEL
LIN {X 0,Y 488.356,Z 685.03,A -85,B 0,C 180,E1 6331.689,E2 6331.689} C_VEL
LIN {X 0,Y 488.265,Z 685.03,A -85,B 0,C 180,E1 6338.179,E2 6338.179} C_VEL
LIN {X 0,Y 488.321,Z 685.03,A -85,B 0,C 180,E1 6344.705,E2 6344.705} C_VEL
LIN {X 0,Y 488.416,Z 685.03,A -85,B 0,C 180,E1 6349.726,E2 6349.726} C_VEL
LIN {X 0,Y 487.774,Z 688.152,A -85,B 0,C 180,E1 6350.901,E2 6350.901} C_VEL
LIN {X 0,Y 487.549,Z 698.573,A -85,B 0,C 180,E1 6352.193,E2 6352.193} C_VEL
LIN {X 0,Y 489.772,Z 705.741,A -85,B 0,C 180,E1 6352.7,E2 6352.7} C_VEL
LIN {X 0,Y 500.963,Z 727.604,A -85,B 0,C 180,E1 6353.866,E2 6353.866} C_VEL
LIN {X 0,Y 499.853,Z 777.364,A -85,B 0,C 180,E1 6354.811,E2 6354.811} C_VEL
LIN {X 0,Y 497.699,Z 816.486,A -85,B 0,C 180,E1 6356.189,E2 6356.189} C_VEL
LIN {X 0,Y 494.766,Z 855.227,A -85,B 0,C 180,E1 6358.257,E2 6358.257} C_VEL
LIN {X 0,Y 491.621,Z 888.216,A -85,B 0,C 180,E1 6360.796,E2 6360.796} C_VEL
LIN {X 0,Y 488.248,Z 920.312,A -85,B 0,C 180,E1 6364.152,E2 6364.152} C_VEL
LIN {X 0,Y 485.5,Z 947.246,A -85,B 0,C 180,E1 6367.861,E2 6367.861} C_VEL
LIN {X 0,Y 483.354,Z 970.605,A -85,B 0,C 180,E1 6372.118,E2 6372.118} C_VEL
LIN {X 0,Y 482.137,Z 988.624,A -85,B 0,C 180,E1 6376.617,E2 6376.617} C_VEL
LIN {X 0,Y 481.649,Z 1000.678,A -85,B 0,C 180,E1 6380.988,E2 6380.988} C_VEL
LIN {X 0,Y 481.415,Z 1006.957,A -85,B 0,C 180,E1 6384.604,E2 6384.604} C_VEL
LIN {X 0,Y 481.429,Z 1010.089,A -85,B 0,C 180,E1 6388.204,E2 6388.204} C_VEL
LIN {X 0,Y 481.49,Z 1010.089,A -85,B 0,C 180,E1 6391.796,E2 6391.796} C_VEL
LIN {X 0,Y 481.555,Z 1005.754,A -85,B 0,C 180,E1 6396.297,E2 6396.297} C_VEL
LIN {X 0,Y 481.72,Z 996.306,A -85,B 0,C 180,E1 6400.833,E2 6400.833} C_VEL
LIN {X 0,Y 482.621,Z 981.29,A -85,B 0,C 180,E1 6405.412,E2 6405.412} C_VEL
LIN {X 0,Y 484.295,Z 959.656,A -85,B 0,C 180,E1 6410.044,E2 6410.044} C_VEL
LIN {X 0,Y 486.848,Z 933.187,A -85,B 0,C 180,E1 6414.202,E2 6414.202} C_VEL
LIN {X 0,Y 489.96,Z 903.786,A -85,B 0,C 180,E1 6417.696,E2 6417.696} C_VEL
LIN {X 0,Y 493.42,Z 870.639,A -85,B 0,C 180,E1 6420.666,E2 6420.666} C_VEL
LIN {X 0,Y 496.255,Z 836.1,A -85,B 0,C 180,E1 6422.86,E2 6422.86} C_VEL
LIN {X 0,Y 498.824,Z 795.942,A -85,B 0,C 180,E1 6424.621,E2 6424.621} C_VEL
LIN {X 0,Y 500.736,Z 756.557,A -85,B 0,C 180,E1 6425.648,E2 6425.648} C_VEL
LIN {X 0,Y 500.275,Z 725.949,A -85,B 0,C 180,E1 6426.209,E2 6426.209} C_VEL
LIN {X 0,Y 480.61,Z 685.03,A -85,B 0,C 180,E1 6428.458,E2 6428.458} C_VEL
LIN {X 0,Y 480.38,Z 685.03,A -85,B 0,C 180,E1 6433.739,E2 6433.739} C_VEL
LIN {X 0,Y 480.462,Z 685.03,A -85,B 0,C 180,E1 6438.918,E2 6438.918} C_VEL
LIN {X 0,Y 480.611,Z 685.03,A -85,B 0,C 180,E1 6444.719,E2 6444.719} C_VEL
LIN {X 0,Y 480.579,Z 685.03,A -85,B 0,C 180,E1 6449.84,E2 6449.84} C_VEL
LIN {X 0,Y 480.554,Z 685.03,A -85,B 0,C 180,E1 6455.905,E2 6455.905} C_VEL
LIN {X 0,Y 480.786,Z 685.03,A -85,B 0,C 180,E1 6461.706,E2 6461.706} C_VEL
LIN {X 0,Y 480.919,Z 685.03,A -85,B 0,C 180,E1 6467.309,E2 6467.309} C_VEL
LIN {X 0,Y 481.037,Z 685.03,A -85,B 0,C 180,E1 6472.789,E2 6472.789} C_VEL
LIN {X 0,Y 481.181,Z 685.03,A -85,B 0,C 180,E1 6478.2,E2 6478.2} C_VEL
LIN {X 0,Y 481.183,Z 685.03,A -85,B 0,C 180,E1 6483.592,E2 6483.592} C_VEL
LIN {X 0,Y 480.978,Z 685.03,A -85,B 0,C 180,E1 6489.021,E2 6489.021} C_VEL
LIN {X 0,Y 480.896,Z 685.03,A -85,B 0,C 180,E1 6494.534,E2 6494.534} C_VEL
LIN {X 0,Y 480.752,Z 685.03,A -85,B 0,C 180,E1 6500.193,E2 6500.193} C_VEL
LIN {X 0,Y 480.612,Z 685.03,A -85,B 0,C 180,E1 6506.07,E2 6506.07} C_VEL
LIN {X 0,Y 480.447,Z 685.03,A -85,B 0,C 180,E1 6512.265,E2 6512.265} C_VEL
LIN {X 0,Y 480.538,Z 685.03,A -85,B 0,C 180,E1 6518.898,E2 6518.898} C_VEL
LIN {X 0,Y 480.438,Z 685.03,A -85,B 0,C 180,E1 6523.747,E2 6523.747} C_VEL
LIN {X 0,Y 480.363,Z 685.03,A -85,B 0,C 180,E1 6528.921,E2 6528.921} C_VEL
LIN {X 0,Y 480.494,Z 685.03,A -85,B 0,C 180,E1 6535.578,E2 6535.578} C_VEL
LIN {X 0,Y 480.695,Z 685.03,A -85,B 0,C 180,E1 6538.35,E2 6538.35} C_VEL
LIN {X 0,Y 491.746,Z 714.218,A -85,B 0,C 180,E1 6540.957,E2 6540.957} C_VEL
LIN {X 0,Y 493.757,Z 728.082,A -85,B 0,C 180,E1 6542.111,E2 6542.111} C_VEL
LIN {X 0,Y 490.39,Z 760.003,A -85,B 0,C 180,E1 6544.701,E2 6544.701} C_VEL
LIN {X 0,Y 487.286,Z 786.911,A -85,B 0,C 180,E1 6547.707,E2 6547.707} C_VEL
LIN {X 0,Y 484.521,Z 811.266,A -85,B 0,C 180,E1 6551.384,E2 6551.384} C_VEL
LIN {X 0,Y 482.637,Z 830.923,A -85,B 0,C 180,E1 6555.515,E2 6555.515} C_VEL
LIN {X 0,Y 481.839,Z 845.755,A -85,B 0,C 180,E1 6559.688,E2 6559.688} C_VEL
LIN {X 0,Y 481.589,Z 855.065,A -85,B 0,C 180,E1 6563.704,E2 6563.704} C_VEL
LIN {X 0,Y 481.447,Z 860.038,A -85,B 0,C 180,E1 6568.204,E2 6568.204} C_VEL
LIN {X 0,Y 481.522,Z 859.987,A -85,B 0,C 180,E1 6571.796,E2 6571.796} C_VEL
LIN {X 0,Y 481.543,Z 854.911,A -85,B 0,C 180,E1 6576.297,E2 6576.297} C_VEL
LIN {X 0,Y 481.82,Z 845.527,A -85,B 0,C 180,E1 6580.301,E2 6580.301} C_VEL
LIN {X 0,Y 482.898,Z 828.702,A -85,B 0,C 180,E1 6584.94,E2 6584.94} C_VEL
LIN {X 0,Y 484.744,Z 809.4,A -85,B 0,C 180,E1 6588.843,E2 6588.843} C_VEL
LIN {X 0,Y 487.59,Z 784.476,A -85,B 0,C 180,E1 6592.518,E2 6592.518} C_VEL
LIN {X 0,Y 491.008,Z 754.45,A -85,B 0,C 180,E1 6595.728,E2 6595.728} C_VEL
LIN {X 0,Y 493.68,Z 722.569,A -85,B 0,C 180,E1 6598.205,E2 6598.205} C_VEL
LIN {X 0,Y 487.864,Z 702.715,A -85,B 0,C 180,E1 6600.011,E2 6600.011} C_VEL
LIN {X 0,Y 480.625,Z 685.03,A -85,B 0,C 180,E1 6601.649,E2 6601.649} C_VEL
LIN {X 0,Y 480.434,Z 685.03,A -85,B 0,C 180,E1 6608.27,E2 6608.27} C_VEL
LIN {X 0,Y 480.413,Z 685.03,A -85,B 0,C 180,E1 6613.753,E2 6613.753} C_VEL
LIN {X 0,Y 480.468,Z 685.03,A -85,B 0,C 180,E1 6618.917,E2 6618.917} C_VEL
LIN {X 0,Y 480.474,Z 685.03,A -85,B 0,C 180,E1 6624.742,E2 6624.742} C_VEL
LIN {X 0,Y 480.497,Z 685.03,A -85,B 0,C 180,E1 6629.842,E2 6629.842} C_VEL
LIN {X 0,Y 480.656,Z 685.03,A -85,B 0,C 180,E1 6635.918,E2 6635.918} C_VEL
LIN {X 0,Y 480.864,Z 685.03,A -85,B 0,C 180,E1 6641.716,E2 6641.716} C_VEL
LIN {X 0,Y 481.034,Z 685.03,A -85,B 0,C 180,E1 6647.32,E2 6647.32} C_VEL
LIN {X 0,Y 481.054,Z 685.03,A -85,B 0,C 180,E1 6652.796,E2 6652.796} C_VEL
LIN {X 0,Y 481.16,Z 685.03,A -85,B 0,C 180,E1 6658.206,E2 6658.206} C_VEL
LIN {X 0,Y 481.186,Z 685.03,A -85,B 0,C 180,E1 6663.599,E2 6663.599} C_VEL
LIN {X 0,Y 480.978,Z 685.03,A -85,B 0,C 180,E1 6669.028,E2 6669.028} C_VEL
LIN {X 0,Y 480.858,Z 685.03,A -85,B 0,C 180,E1 6674.542,E2 6674.542} C_VEL
LIN {X 0,Y 480.729,Z 685.03,A -85,B 0,C 180,E1 6680.201,E2 6680.201} C_VEL
LIN {X 0,Y 480.601,Z 685.03,A -85,B 0,C 180,E1 6686.078,E2 6686.078} C_VEL
LIN {X 0,Y 480.407,Z 685.03,A -85,B 0,C 180,E1 6692.276,E2 6692.276} C_VEL
LIN {X 0,Y 480.329,Z 685.03,A -85,B 0,C 180,E1 6698.927,E2 6698.927} C_VEL
LIN {X 0,Y 480.353,Z 685.03,A -85,B 0,C 180,E1 6703.736,E2 6703.736} C_VEL
LIN {X 0,Y 480.424,Z 685.03,A -85,B 0,C 180,E1 6709.727,E2 6709.727} C_VEL
LIN {X 0,Y 480.611,Z 685.031,A -85,B 0,C 180,E1 6711.629,E2 6711.629} C_VEL
LIN {X 0,Y 489.772,Z 705.741,A -85,B 0,C 180,E1 6712.7,E2 6712.7} C_VEL
LIN {X 0,Y 493.409,Z 717.782,A -85,B 0,C 180,E1 6713.167,E2 6713.167} C_VEL
LIN {X 0,Y 494.071,Z 739.967,A -85,B 0,C 180,E1 6713.589,E2 6713.589} C_VEL
LIN {X 0,Y 492.614,Z 783.659,A -85,B 0,C 180,E1 6714.543,E2 6714.543} C_VEL
LIN {X 0,Y 490.109,Z 823.573,A -85,B 0,C 180,E1 6716.106,E2 6716.106} C_VEL
LIN {X 0,Y 486.759,Z 863.786,A -85,B 0,C 180,E1 6718.468,E2 6718.468} C_VEL
LIN {X 0,Y 483.493,Z 897.656,A -85,B 0,C 180,E1 6721.227,E2 6721.227} C_VEL
LIN {X 0,Y 479.895,Z 929.366,A -85,B 0,C 180,E1 6724.881,E2 6724.881} C_VEL
LIN {X 0,Y 477.046,Z 955.426,A -85,B 0,C 180,E1 6728.863,E2 6728.863} C_VEL
LIN {X 0,Y 475.105,Z 976.238,A -85,B 0,C 180,E1 6733.084,E2 6733.084} C_VEL
LIN {X 0,Y 474.043,Z 992.402,A -85,B 0,C 180,E1 6737.592,E2 6737.592} C_VEL
LIN {X 0,Y 473.686,Z 1002.627,A -85,B 0,C 180,E1 6741.773,E2 6741.773} C_VEL
LIN {X 0,Y 473.509,Z 1008.909,A -85,B 0,C 180,E1 6746.346,E2 6746.346} C_VEL
LIN {X 0,Y 473.544,Z 1010.5,A -85,B 0,C 180,E1 6750,E2 6750} C_VEL
LIN {X 0,Y 473.482,Z 1008.911,A -85,B 0,C 180,E1 6753.655,E2 6753.655} C_VEL
LIN {X 0,Y 473.71,Z 1002.625,A -85,B 0,C 180,E1 6758.228,E2 6758.228} C_VEL
LIN {X 0,Y 474.313,Z 989.985,A -85,B 0,C 180,E1 6763.191,E2 6763.191} C_VEL
LIN {X 0,Y 475.516,Z 972.248,A -85,B 0,C 180,E1 6767.824,E2 6767.824} C_VEL
LIN {X 0,Y 477.624,Z 950.187,A -85,B 0,C 180,E1 6772.029,E2 6772.029} C_VEL
LIN {X 0,Y 480.497,Z 923.858,A -85,B 0,C 180,E1 6775.832,E2 6775.832} C_VEL
LIN {X 0,Y 483.907,Z 894.233,A -85,B 0,C 180,E1 6779.09,E2 6779.09} C_VEL
LIN {X 0,Y 487.092,Z 860.127,A -85,B 0,C 180,E1 6781.78,E2 6781.78} C_VEL
LIN {X 0,Y 490.141,Z 822.127,A -85,B 0,C 180,E1 6783.965,E2 6783.965} C_VEL
LIN {X 0,Y 492.749,Z 781.817,A -85,B 0,C 180,E1 6785.507,E2 6785.507} C_VEL
LIN {X 0,Y 494.212,Z 739.519,A -85,B 0,C 180,E1 6786.409,E2 6786.409} C_VEL
LIN {X 0,Y 493.597,Z 728.868,A -85,B 0,C 180,E1 6786.634,E2 6786.634} C_VEL
LIN {X 0,Y 472.659,Z 685.03,A -85,B 0,C 180,E1 6789.07,E2 6789.07} C_VEL
LIN {X 0,Y 472.401,Z 685.03,A -85,B 0,C 180,E1 6795.351,E2 6795.351} C_VEL
LIN {X 0,Y 472.556,Z 685.03,A -85,B 0,C 180,E1 6800.308,E2 6800.308} C_VEL
LIN {X 0,Y 472.666,Z 685.03,A -85,B 0,C 180,E1 6806.104,E2 6806.104} C_VEL
LIN {X 0,Y 472.606,Z 685.03,A -85,B 0,C 180,E1 6811.382,E2 6811.382} C_VEL
LIN {X 0,Y 472.714,Z 685.03,A -85,B 0,C 180,E1 6817.779,E2 6817.779} C_VEL
LIN {X 0,Y 472.917,Z 685.03,A -85,B 0,C 180,E1 6823.309,E2 6823.309} C_VEL
LIN {X 0,Y 473.009,Z 685.03,A -85,B 0,C 180,E1 6828.962,E2 6828.962} C_VEL
LIN {X 0,Y 473.229,Z 685.03,A -85,B 0,C 180,E1 6834.508,E2 6834.508} C_VEL
LIN {X 0,Y 473.36,Z 685.03,A -85,B 0,C 180,E1 6839.997,E2 6839.997} C_VEL
LIN {X 0,Y 473.244,Z 685.03,A -85,B 0,C 180,E1 6845.485,E2 6845.485} C_VEL
LIN {X 0,Y 473.021,Z 685.03,A -85,B 0,C 180,E1 6851.031,E2 6851.031} C_VEL
LIN {X 0,Y 472.886,Z 685.03,A -85,B 0,C 180,E1 6856.802,E2 6856.802} C_VEL
LIN {X 0,Y 472.787,Z 685.03,A -85,B 0,C 180,E1 6862.514,E2 6862.514} C_VEL
LIN {X 0,Y 472.558,Z 685.03,A -85,B 0,C 180,E1 6868.613,E2 6868.613} C_VEL
LIN {X 0,Y 472.56,Z 685.03,A -85,B 0,C 180,E1 6875.077,E2 6875.077} C_VEL
LIN {X 0,Y 472.517,Z 685.03,A -85,B 0,C 180,E1 6879.964,E2 6879.964} C_VEL
LIN {X 0,Y 472.423,Z 685.03,A -85,B 0,C 180,E1 6885.355,E2 6885.355} C_VEL
LIN {X 0,Y 472.526,Z 685.03,A -85,B 0,C 180,E1 6892.645,E2 6892.645} C_VEL
LIN {X 0,Y 472.757,Z 685.836,A -85,B 0,C 180,E1 6897.667,E2 6897.667} C_VEL
LIN {X 0,Y 484.84,Z 715.543,A -85,B 0,C 180,E1 6900.409,E2 6900.409} C_VEL
LIN {X 0,Y 487.157,Z 729.666,A -85,B 0,C 180,E1 6901.638,E2 6901.638} C_VEL
LIN {X 0,Y 483.78,Z 759.847,A -85,B 0,C 180,E1 6904.108,E2 6904.108} C_VEL
LIN {X 0,Y 480.458,Z 786.878,A -85,B 0,C 180,E1 6907.129,E2 6907.129} C_VEL
LIN {X 0,Y 477.326,Z 811.54,A -85,B 0,C 180,E1 6910.853,E2 6910.853} C_VEL
LIN {X 0,Y 475.3,Z 830.607,A -85,B 0,C 180,E1 6914.816,E2 6914.816} C_VEL
LIN {X 0,Y 474.073,Z 844.793,A -85,B 0,C 180,E1 6918.99,E2 6918.99} C_VEL
LIN {X 0,Y 473.684,Z 855.064,A -85,B 0,C 180,E1 6923.598,E2 6923.598} C_VEL
LIN {X 0,Y 473.545,Z 860.037,A -85,B 0,C 180,E1 6928.174,E2 6928.174} C_VEL
LIN {X 0,Y 473.618,Z 859.987,A -85,B 0,C 180,E1 6931.826,E2 6931.826} C_VEL
LIN {X 0,Y 473.643,Z 854.913,A -85,B 0,C 180,E1 6936.402,E2 6936.402} C_VEL
LIN {X 0,Y 474.238,Z 843.182,A -85,B 0,C 180,E1 6941.471,E2 6941.471} C_VEL
LIN {X 0,Y 475.542,Z 828.238,A -85,B 0,C 180,E1 6945.648,E2 6945.648} C_VEL
LIN {X 0,Y 477.944,Z 806.985,A -85,B 0,C 180,E1 6949.841,E2 6949.841} C_VEL
LIN {X 0,Y 480.907,Z 782.579,A -85,B 0,C 180,E1 6953.338,E2 6953.338} C_VEL
LIN {X 0,Y 484.487,Z 753.342,A -85,B 0,C 180,E1 6956.407,E2 6956.407} C_VEL
LIN {X 0,Y 487.08,Z 725.385,A -85,B 0,C 180,E1 6958.597,E2 6958.597} C_VEL
LIN {X 0,Y 481.103,Z 705.384,A -85,B 0,C 180,E1 6960.479,E2 6960.479} C_VEL
LIN {X 0,Y 472.694,Z 685.03,A -85,B 0,C 180,E1 6962.33,E2 6962.33} C_VEL
LIN {X 0,Y 472.533,Z 685.03,A -85,B 0,C 180,E1 6967.355,E2 6967.355} C_VEL
LIN {X 0,Y 472.441,Z 685.03,A -85,B 0,C 180,E1 6974.643,E2 6974.643} C_VEL
LIN {X 0,Y 472.537,Z 685.03,A -85,B 0,C 180,E1 6980.315,E2 6980.315} C_VEL
LIN {X 0,Y 472.517,Z 685.03,A -85,B 0,C 180,E1 6986.131,E2 6986.131} C_VEL
LIN {X 0,Y 472.611,Z 685.03,A -85,B 0,C 180,E1 6991.391,E2 6991.391} C_VEL
LIN {X 0,Y 472.838,Z 685.03,A -85,B 0,C 180,E1 6997.743,E2 6997.743} C_VEL
LIN {X 0,Y 472.997,Z 685.03,A -85,B 0,C 180,E1 7003.319,E2 7003.319} C_VEL
LIN {X 0,Y 473.114,Z 685.03,A -85,B 0,C 180,E1 7008.972,E2 7008.972} C_VEL
LIN {X 0,Y 473.23,Z 685.03,A -85,B 0,C 180,E1 7014.515,E2 7014.515} C_VEL
LIN {X 0,Y 473.362,Z 685.03,A -85,B 0,C 180,E1 7020.003,E2 7020.003} C_VEL
LIN {X 0,Y 473.245,Z 685.03,A -85,B 0,C 180,E1 7025.492,E2 7025.492} C_VEL
LIN {X 0,Y 473.018,Z 685.03,A -85,B 0,C 180,E1 7031.038,E2 7031.038} C_VEL
LIN {X 0,Y 472.879,Z 685.03,A -85,B 0,C 180,E1 7036.8,E2 7036.8} C_VEL
LIN {X 0,Y 472.706,Z 685.03,A -85,B 0,C 180,E1 7042.526,E2 7042.526} C_VEL
LIN {X 0,Y 472.559,Z 685.03,A -85,B 0,C 180,E1 7048.621,E2 7048.621} C_VEL
LIN {X 0,Y 472.447,Z 685.03,A -85,B 0,C 180,E1 7055.095,E2 7055.095} C_VEL
LIN {X 0,Y 472.348,Z 685.03,A -85,B 0,C 180,E1 7062.136,E2 7062.136} C_VEL
LIN {X 0,Y 472.426,Z 685.03,A -85,B 0,C 180,E1 7067.874,E2 7067.874} C_VEL
LIN {X 0,Y 472.702,Z 685.549,A -85,B 0,C 180,E1 7070.991,E2 7070.991} C_VEL
LIN {X 0,Y 493.975,Z 729.56,A -85,B 0,C 180,E1 7073.407,E2 7073.407} C_VEL
LIN {X 0,Y 494.071,Z 739.967,A -85,B 0,C 180,E1 7073.589,E2 7073.589} C_VEL
LIN {X 0,Y 490.314,Z 757.117,A -85,B 0,C 180,E1 7073.646,E2 7073.646} C_VEL
LIN {X 0,Y 486.243,Z 774.082,A -85,B 0,C 180,E1 7073.813,E2 7073.813} C_VEL
LIN {X 0,Y 483.703,Z 813.85,A -85,B 0,C 180,E1 7075.228,E2 7075.228} C_VEL
LIN {X 0,Y 480.423,Z 852.664,A -85,B 0,C 180,E1 7077.351,E2 7077.351} C_VEL
LIN {X 0,Y 476.931,Z 888.536,A -85,B 0,C 180,E1 7080.081,E2 7080.081} C_VEL
LIN {X 0,Y 473.667,Z 920.051,A -85,B 0,C 180,E1 7083.271,E2 7083.271} C_VEL
LIN {X 0,Y 470.412,Z 947.511,A -85,B 0,C 180,E1 7087.157,E2 7087.157} C_VEL
LIN {X 0,Y 468.153,Z 969.18,A -85,B 0,C 180,E1 7091.196,E2 7091.196} C_VEL
LIN {X 0,Y 466.572,Z 988.073,A -85,B 0,C 180,E1 7095.99,E2 7095.99} C_VEL
LIN {X 0,Y 465.91,Z 1000.678,A -85,B 0,C 180,E1 7100.68,E2 7100.68} C_VEL
LIN {X 0,Y 465.641,Z 1006.956,A -85,B 0,C 180,E1 7104.421,E2 7104.421} C_VEL
LIN {X 0,Y 465.626,Z 1010.089,A -85,B 0,C 180,E1 7108.143,E2 7108.143} C_VEL
LIN {X 0,Y 465.677,Z 1010.09,A -85,B 0,C 180,E1 7111.857,E2 7111.857} C_VEL
LIN {X 0,Y 465.74,Z 1005.754,A -85,B 0,C 180,E1 7116.511,E2 7116.511} C_VEL
LIN {X 0,Y 466.024,Z 996.306,A -85,B 0,C 180,E1 7121.203,E2 7121.203} C_VEL
LIN {X 0,Y 467.086,Z 981.292,A -85,B 0,C 180,E1 7125.938,E2 7125.938} C_VEL
LIN {X 0,Y 469.092,Z 959.653,A -85,B 0,C 180,E1 7130.723,E2 7130.723} C_VEL
LIN {X 0,Y 471.902,Z 934.604,A -85,B 0,C 180,E1 7134.815,E2 7134.815} C_VEL
LIN {X 0,Y 474.88,Z 908.519,A -85,B 0,C 180,E1 7138.011,E2 7138.011} C_VEL
LIN {X 0,Y 478.677,Z 871.314,A -85,B 0,C 180,E1 7141.334,E2 7141.334} C_VEL
LIN {X 0,Y 482.145,Z 833.224,A -85,B 0,C 180,E1 7143.809,E2 7143.809} C_VEL
LIN {X 0,Y 484.983,Z 794.446,A -85,B 0,C 180,E1 7145.552,E2 7145.552} C_VEL
LIN {X 0,Y 487.195,Z 753.689,A -85,B 0,C 180,E1 7146.64,E2 7146.64} C_VEL
LIN {X 0,Y 486.961,Z 731.661,A -85,B 0,C 180,E1 7147.066,E2 7147.066} C_VEL
LIN {X 0,Y 464.669,Z 685.03,A -85,B 0,C 180,E1 7149.748,E2 7149.748} C_VEL
LIN {X 0,Y 464.481,Z 685.03,A -85,B 0,C 180,E1 7155.621,E2 7155.621} C_VEL
LIN {X 0,Y 464.66,Z 685.03,A -85,B 0,C 180,E1 7161.899,E2 7161.899} C_VEL
LIN {X 0,Y 464.708,Z 685.03,A -85,B 0,C 180,E1 7167.594,E2 7167.594} C_VEL
LIN {X 0,Y 464.677,Z 685.03,A -85,B 0,C 180,E1 7172.957,E2 7172.957} C_VEL
LIN {X 0,Y 464.845,Z 685.03,A -85,B 0,C 180,E1 7179.077,E2 7179.077} C_VEL
LIN {X 0,Y 465.051,Z 685.03,A -85,B 0,C 180,E1 7184.952,E2 7184.952} C_VEL
LIN {X 0,Y 465.195,Z 685.03,A -85,B 0,C 180,E1 7190.663,E2 7190.663} C_VEL
LIN {X 0,Y 465.479,Z 685.03,A -85,B 0,C 180,E1 7196.279,E2 7196.279} C_VEL
LIN {X 0,Y 465.602,Z 685.03,A -85,B 0,C 180,E1 7201.854,E2 7201.854} C_VEL
LIN {X 0,Y 465.278,Z 685.03,A -85,B 0,C 180,E1 7207.45,E2 7207.45} C_VEL
LIN {X 0,Y 465.102,Z 685.03,A -85,B 0,C 180,E1 7213.262,E2 7213.262} C_VEL
LIN {X 0,Y 464.869,Z 685.03,A -85,B 0,C 180,E1 7219.719,E2 7219.719} C_VEL
LIN {X 0,Y 464.762,Z 685.03,A -85,B 0,C 180,E1 7224.96,E2 7224.96} C_VEL
LIN {X 0,Y 464.522,Z 685.03,A -85,B 0,C 180,E1 7231.309,E2 7231.309} C_VEL
LIN {X 0,Y 464.598,Z 685.03,A -85,B 0,C 180,E1 7238.098,E2 7238.098} C_VEL
LIN {X 0,Y 464.516,Z 685.03,A -85,B 0,C 180,E1 7244.383,E2 7244.383} C_VEL
LIN {X 0,Y 464.469,Z 685.03,A -85,B 0,C 180,E1 7251.224,E2 7251.224} C_VEL
LIN {X 0,Y 464.718,Z 685.253,A -85,B 0,C 180,E1 7256.885,E2 7256.885} C_VEL
LIN {X 0,Y 477.793,Z 717.083,A -85,B 0,C 180,E1 7259.861,E2 7259.861} C_VEL
LIN {X 0,Y 480.573,Z 731.522,A -85,B 0,C 180,E1 7261.174,E2 7261.174} C_VEL
LIN {X 0,Y 476.954,Z 761.916,A -85,B 0,C 180,E1 7263.709,E2 7263.709} C_VEL
LIN {X 0,Y 473.378,Z 788.677,A -85,B 0,C 180,E1 7266.767,E2 7266.767} C_VEL
LIN {X 0,Y 470.031,Z 813.148,A -85,B 0,C 180,E1 7270.544,E2 7270.544} C_VEL
LIN {X 0,Y 467.781,Z 832.106,A -85,B 0,C 180,E1 7274.566,E2 7274.566} C_VEL
LIN {X 0,Y 466.348,Z 847.42,A -85,B 0,C 180,E1 7279.277,E2 7279.277} C_VEL
LIN {X 0,Y 465.882,Z 856.031,A -85,B 0,C 180,E1 7283.491,E2 7283.491} C_VEL
LIN {X 0,Y 465.673,Z 860.555,A -85,B 0,C 180,E1 7288.143,E2 7288.143} C_VEL
LIN {X 0,Y 465.737,Z 860.499,A -85,B 0,C 180,E1 7291.857,E2 7291.857} C_VEL
LIN {X 0,Y 465.848,Z 855.901,A -85,B 0,C 180,E1 7296.51,E2 7296.51} C_VEL
LIN {X 0,Y 466.452,Z 845.972,A -85,B 0,C 180,E1 7301.192,E2 7301.192} C_VEL
LIN {X 0,Y 467.871,Z 831.728,A -85,B 0,C 180,E1 7305.431,E2 7305.431} C_VEL
LIN {X 0,Y 470.297,Z 811.301,A -85,B 0,C 180,E1 7309.688,E2 7309.688} C_VEL
LIN {X 0,Y 473.626,Z 786.292,A -85,B 0,C 180,E1 7313.469,E2 7313.469} C_VEL
LIN {X 0,Y 477.473,Z 757.404,A -85,B 0,C 180,E1 7316.64,E2 7316.64} C_VEL
LIN {X 0,Y 480.411,Z 727.718,A -85,B 0,C 180,E1 7319.045,E2 7319.045} C_VEL
LIN {X 0,Y 474.629,Z 708.72,A -85,B 0,C 180,E1 7320.875,E2 7320.875} C_VEL
LIN {X 0,Y 464.681,Z 685.03,A -85,B 0,C 180,E1 7323.078,E2 7323.078} C_VEL
LIN {X 0,Y 464.484,Z 685.03,A -85,B 0,C 180,E1 7328.778,E2 7328.778} C_VEL
LIN {X 0,Y 464.525,Z 685.03,A -85,B 0,C 180,E1 7335.615,E2 7335.615} C_VEL
LIN {X 0,Y 464.607,Z 685.03,A -85,B 0,C 180,E1 7341.903,E2 7341.903} C_VEL
LIN {X 0,Y 464.592,Z 685.03,A -85,B 0,C 180,E1 7348.696,E2 7348.696} C_VEL
LIN {X 0,Y 464.827,Z 685.03,A -85,B 0,C 180,E1 7355.364,E2 7355.364} C_VEL
LIN {X 0,Y 464.983,Z 685.03,A -85,B 0,C 180,E1 7361.068,E2 7361.068} C_VEL
LIN {X 0,Y 465.206,Z 685.03,A -85,B 0,C 180,E1 7366.881,E2 7366.881} C_VEL
LIN {X 0,Y 465.241,Z 685.03,A -85,B 0,C 180,E1 7372.675,E2 7372.675} C_VEL
LIN {X 0,Y 465.388,Z 685.03,A -85,B 0,C 180,E1 7378.146,E2 7378.146} C_VEL
LIN {X 0,Y 465.389,Z 685.03,A -85,B 0,C 180,E1 7383.721,E2 7383.721} C_VEL
LIN {X 0,Y 465.139,Z 685.03,A -85,B 0,C 180,E1 7389.338,E2 7389.338} C_VEL
LIN {X 0,Y 464.993,Z 685.03,A -85,B 0,C 180,E1 7395.05,E2 7395.05} C_VEL
LIN {X 0,Y 464.864,Z 685.03,A -85,B 0,C 180,E1 7400.923,E2 7400.923} C_VEL
LIN {X 0,Y 464.697,Z 685.03,A -85,B 0,C 180,E1 7407.042,E2 7407.042} C_VEL
LIN {X 0,Y 464.512,Z 685.03,A -85,B 0,C 180,E1 7413.523,E2 7413.523} C_VEL
LIN {X 0,Y 464.403,Z 685.03,A -85,B 0,C 180,E1 7420.532,E2 7420.532} C_VEL
LIN {X 0,Y 464.519,Z 685.03,A -85,B 0,C 180,E1 7426.985,E2 7426.985} C_VEL
LIN {X 0,Y 464.694,Z 685.443,A -85,B 0,C 180,E1 7430.291,E2 7430.291} C_VEL
LIN {X 0,Y 487.378,Z 732.569,A -85,B 0,C 180,E1 7432.986,E2 7432.986} C_VEL
LIN {X 0,Y 486.243,Z 774.082,A -85,B 0,C 180,E1 7433.813,E2 7433.813} C_VEL
LIN {X 0,Y 481.607,Z 790.856,A -85,B 0,C 180,E1 7434.09,E2 7434.09} C_VEL
LIN {X 0,Y 477.31,Z 805.328,A -85,B 0,C 180,E1 7434.428,E2 7434.428} C_VEL
LIN {X 0,Y 477.092,Z 807.406,A -85,B 0,C 180,E1 7434.51,E2 7434.51} C_VEL
LIN {X 0,Y 473.592,Z 848.292,A -85,B 0,C 180,E1 7436.669,E2 7436.669} C_VEL
LIN {X 0,Y 469.844,Z 885.166,A -85,B 0,C 180,E1 7439.455,E2 7439.455} C_VEL
LIN {X 0,Y 466.177,Z 918.531,A -85,B 0,C 180,E1 7442.829,E2 7442.829} C_VEL
LIN {X 0,Y 463.241,Z 944.822,A -85,B 0,C 180,E1 7446.316,E2 7446.316} C_VEL
LIN {X 0,Y 460.505,Z 969.179,A -85,B 0,C 180,E1 7450.872,E2 7450.872} C_VEL
LIN {X 0,Y 458.765,Z 988.072,A -85,B 0,C 180,E1 7455.747,E2 7455.747} C_VEL
LIN {X 0,Y 458.033,Z 1000.678,A -85,B 0,C 180,E1 7460.519,E2 7460.519} C_VEL
LIN {X 0,Y 457.748,Z 1006.955,A -85,B 0,C 180,E1 7464.324,E2 7464.324} C_VEL
LIN {X 0,Y 457.722,Z 1010.089,A -85,B 0,C 180,E1 7468.111,E2 7468.111} C_VEL
LIN {X 0,Y 457.771,Z 1010.09,A -85,B 0,C 180,E1 7471.889,E2 7471.889} C_VEL
LIN {X 0,Y 457.849,Z 1005.754,A -85,B 0,C 180,E1 7476.624,E2 7476.624} C_VEL
LIN {X 0,Y 458.194,Z 996.307,A -85,B 0,C 180,E1 7481.397,E2 7481.397} C_VEL
LIN {X 0,Y 459.331,Z 981.292,A -85,B 0,C 180,E1 7486.215,E2 7486.215} C_VEL
LIN {X 0,Y 461.488,Z 959.651,A -85,B 0,C 180,E1 7491.081,E2 7491.081} C_VEL
LIN {X 0,Y 464.245,Z 935.926,A -85,B 0,C 180,E1 7494.996,E2 7494.996} C_VEL
LIN {X 0,Y 467.855,Z 903.547,A -85,B 0,C 180,E1 7498.802,E2 7498.802} C_VEL
LIN {X 0,Y 471.611,Z 868.199,A -85,B 0,C 180,E1 7501.928,E2 7501.928} C_VEL
LIN {X 0,Y 475.17,Z 830.996,A -85,B 0,C 180,E1 7504.343,E2 7504.343} C_VEL
LIN {X 0,Y 478.283,Z 790.722,A -85,B 0,C 180,E1 7506.135,E2 7506.135} C_VEL
LIN {X 0,Y 480.494,Z 751.185,A -85,B 0,C 180,E1 7507.174,E2 7507.174} C_VEL
LIN {X 0,Y 480.307,Z 734.508,A -85,B 0,C 180,E1 7507.506,E2 7507.506} C_VEL
LIN {X 0,Y 456.665,Z 685.03,A -85,B 0,C 180,E1 7510.535,E2 7510.535} C_VEL
LIN {X 0,Y 456.591,Z 685.03,A -85,B 0,C 180,E1 7516.642,E2 7516.642} C_VEL
LIN {X 0,Y 456.733,Z 685.03,A -85,B 0,C 180,E1 7522.46,E2 7522.46} C_VEL
LIN {X 0,Y 456.783,Z 685.03,A -85,B 0,C 180,E1 7528.09,E2 7528.09} C_VEL
LIN {X 0,Y 456.744,Z 685.03,A -85,B 0,C 180,E1 7534.563,E2 7534.563} C_VEL
LIN {X 0,Y 456.977,Z 685.03,A -85,B 0,C 180,E1 7540.716,E2 7540.716} C_VEL
LIN {X 0,Y 457.219,Z 685.03,A -85,B 0,C 180,E1 7546.64,E2 7546.64} C_VEL
LIN {X 0,Y 457.312,Z 685.03,A -85,B 0,C 180,E1 7552.412,E2 7552.412} C_VEL
LIN {X 0,Y 457.505,Z 685.03,A -85,B 0,C 180,E1 7558.106,E2 7558.106} C_VEL
LIN {X 0,Y 457.477,Z 685.03,A -85,B 0,C 180,E1 7563.779,E2 7563.779} C_VEL
LIN {X 0,Y 457.234,Z 685.03,A -85,B 0,C 180,E1 7569.494,E2 7569.494} C_VEL
LIN {X 0,Y 457.084,Z 685.03,A -85,B 0,C 180,E1 7575.309,E2 7575.309} C_VEL
LIN {X 0,Y 456.943,Z 685.03,A -85,B 0,C 180,E1 7581.295,E2 7581.295} C_VEL
LIN {X 0,Y 456.753,Z 685.03,A -85,B 0,C 180,E1 7587.544,E2 7587.544} C_VEL
LIN {X 0,Y 456.607,Z 685.03,A -85,B 0,C 180,E1 7594.29,E2 7594.29} C_VEL
LIN {X 0,Y 456.66,Z 685.03,A -85,B 0,C 180,E1 7600.535,E2 7600.535} C_VEL
LIN {X 0,Y 456.574,Z 685.03,A -85,B 0,C 180,E1 7606.635,E2 7606.635} C_VEL
LIN {X 0,Y 456.59,Z 685.03,A -85,B 0,C 180,E1 7613.496,E2 7613.496} C_VEL
LIN {X 0,Y 456.719,Z 685.15,A -85,B 0,C 180,E1 7616.098,E2 7616.098} C_VEL
LIN {X 0,Y 469.788,Z 716.32,A -85,B 0,C 180,E1 7619.074,E2 7619.074} C_VEL
LIN {X 0,Y 473.997,Z 732.933,A -85,B 0,C 180,E1 7620.678,E2 7620.678} C_VEL
LIN {X 0,Y 470.251,Z 762.982,A -85,B 0,C 180,E1 7623.195,E2 7623.195} C_VEL
LIN {X 0,Y 466.348,Z 790.536,A -85,B 0,C 180,E1 7626.395,E2 7626.395} C_VEL
LIN {X 0,Y 462.748,Z 814.785,A -85,B 0,C 180,E1 7630.225,E2 7630.225} C_VEL
LIN {X 0,Y 460.262,Z 833.603,A -85,B 0,C 180,E1 7634.307,E2 7634.307} C_VEL
LIN {X 0,Y 458.678,Z 848.826,A -85,B 0,C 180,E1 7639.096,E2 7639.096} C_VEL
LIN {X 0,Y 458.124,Z 857.385,A -85,B 0,C 180,E1 7643.38,E2 7643.38} C_VEL
LIN {X 0,Y 457.914,Z 861.866,A -85,B 0,C 180,E1 7648.112,E2 7648.112} C_VEL
LIN {X 0,Y 457.976,Z 861.81,A -85,B 0,C 180,E1 7651.888,E2 7651.888} C_VEL
LIN {X 0,Y 458.094,Z 857.253,A -85,B 0,C 180,E1 7656.62,E2 7656.62} C_VEL
LIN {X 0,Y 458.805,Z 847.382,A -85,B 0,C 180,E1 7661.381,E2 7661.381} C_VEL
LIN {X 0,Y 460.571,Z 831.268,A -85,B 0,C 180,E1 7666.17,E2 7666.17} C_VEL
LIN {X 0,Y 463.426,Z 810.29,A -85,B 0,C 180,E1 7670.49,E2 7670.49} C_VEL
LIN {X 0,Y 467.211,Z 784.436,A -85,B 0,C 180,E1 7674.318,E2 7674.318} C_VEL
LIN {X 0,Y 471.211,Z 755.422,A -85,B 0,C 180,E1 7677.431,E2 7677.431} C_VEL
LIN {X 0,Y 473.84,Z 730.796,A -85,B 0,C 180,E1 7679.419,E2 7679.419} C_VEL
LIN {X 0,Y 467.626,Z 710.983,A -85,B 0,C 180,E1 7681.388,E2 7681.388} C_VEL
LIN {X 0,Y 456.692,Z 685.03,A -85,B 0,C 180,E1 7683.904,E2 7683.904} C_VEL
LIN {X 0,Y 456.571,Z 685.03,A -85,B 0,C 180,E1 7690.532,E2 7690.532} C_VEL
LIN {X 0,Y 456.655,Z 685.03,A -85,B 0,C 180,E1 7696.634,E2 7696.634} C_VEL
LIN {X 0,Y 456.667,Z 685.03,A -85,B 0,C 180,E1 7702.471,E2 7702.471} C_VEL
LIN {X 0,Y 456.646,Z 685.03,A -85,B 0,C 180,E1 7709.224,E2 7709.224} C_VEL
LIN {X 0,Y 456.821,Z 685.03,A -85,B 0,C 180,E1 7714.575,E2 7714.575} C_VEL
LIN {X 0,Y 457.056,Z 685.03,A -85,B 0,C 180,E1 7720.727,E2 7720.727} C_VEL
LIN {X 0,Y 457.304,Z 685.03,A -85,B 0,C 180,E1 7726.65,E2 7726.65} C_VEL
LIN {X 0,Y 457.316,Z 685.03,A -85,B 0,C 180,E1 7732.669,E2 7732.669} C_VEL
LIN {X 0,Y 457.485,Z 685.03,A -85,B 0,C 180,E1 7738.114,E2 7738.114} C_VEL
LIN {X 0,Y 457.48,Z 685.03,A -85,B 0,C 180,E1 7743.786,E2 7743.786} C_VEL
LIN {X 0,Y 457.236,Z 685.03,A -85,B 0,C 180,E1 7749.501,E2 7749.501} C_VEL
LIN {X 0,Y 457.059,Z 685.03,A -85,B 0,C 180,E1 7755.317,E2 7755.317} C_VEL
LIN {X 0,Y 456.899,Z 685.03,A -85,B 0,C 180,E1 7761.305,E2 7761.305} C_VEL
LIN {X 0,Y 456.759,Z 685.03,A -85,B 0,C 180,E1 7767.552,E2 7767.552} C_VEL
LIN {X 0,Y 456.535,Z 685.03,A -85,B 0,C 180,E1 7774.277,E2 7774.277} C_VEL
LIN {X 0,Y 456.52,Z 685.03,A -85,B 0,C 180,E1 7780.514,E2 7780.514} C_VEL
LIN {X 0,Y 456.586,Z 685.03,A -85,B 0,C 180,E1 7786.644,E2 7786.644} C_VEL
LIN {X 0,Y 456.677,Z 685.03,A -85,B 0,C 180,E1 7789.537,E2 7789.537} C_VEL
LIN {X 0,Y 480.666,Z 736.641,A -85,B 0,C 180,E1 7792.562,E2 7792.562} C_VEL
LIN {X 0,Y 479.1,Z 779.797,A -85,B 0,C 180,E1 7793.517,E2 7793.517} C_VEL
LIN {X 0,Y 477.092,Z 807.406,A -85,B 0,C 180,E1 7794.51,E2 7794.51} C_VEL
LIN {X 0,Y 472.412,Z 823.684,A -85,B 0,C 180,E1 7795.061,E2 7795.061} C_VEL
LIN {X 0,Y 467.253,Z 839.531,A -85,B 0,C 180,E1 7795.736,E2 7795.736} C_VEL
LIN {X 0,Y 463.399,Z 876.204,A -85,B 0,C 180,E1 7798.348,E2 7798.348} C_VEL
LIN {X 0,Y 459.572,Z 909.709,A -85,B 0,C 180,E1 7801.569,E2 7801.569} C_VEL
LIN {X 0,Y 456.01,Z 940.055,A -85,B 0,C 180,E1 7805.408,E2 7805.408} C_VEL
LIN {X 0,Y 453.484,Z 962.302,A -85,B 0,C 180,E1 7809.084,E2 7809.084} C_VEL
LIN {X 0,Y 451.452,Z 981.289,A -85,B 0,C 180,E1 7813.494,E2 7813.494} C_VEL
LIN {X 0,Y 450.357,Z 996.307,A -85,B 0,C 180,E1 7818.402,E2 7818.402} C_VEL
LIN {X 0,Y 449.957,Z 1005.749,A -85,B 0,C 180,E1 7823.259,E2 7823.259} C_VEL
LIN {X 0,Y 449.84,Z 1010.089,A -85,B 0,C 180,E1 7828.078,E2 7828.078} C_VEL
LIN {X 0,Y 449.884,Z 1010.09,A -85,B 0,C 180,E1 7831.922,E2 7831.922} C_VEL
LIN {X 0,Y 449.945,Z 1005.754,A -85,B 0,C 180,E1 7836.741,E2 7836.741} C_VEL
LIN {X 0,Y 450.341,Z 996.307,A -85,B 0,C 180,E1 7841.598,E2 7841.598} C_VEL
LIN {X 0,Y 451.568,Z 981.292,A -85,B 0,C 180,E1 7846.502,E2 7846.502} C_VEL
LIN {X 0,Y 453.777,Z 960.596,A -85,B 0,C 180,E1 7851.254,E2 7851.254} C_VEL
LIN {X 0,Y 456.733,Z 934.137,A -85,B 0,C 180,E1 7855.436,E2 7855.436} C_VEL
LIN {X 0,Y 460.522,Z 901.538,A -85,B 0,C 180,E1 7859.305,E2 7859.305} C_VEL
LIN {X 0,Y 464.41,Z 866.755,A -85,B 0,C 180,E1 7862.407,E2 7862.407} C_VEL
LIN {X 0,Y 468.169,Z 829.613,A -85,B 0,C 180,E1 7864.838,E2 7864.838} C_VEL
LIN {X 0,Y 471.414,Z 790.318,A -85,B 0,C 180,E1 7866.615,E2 7866.615} C_VEL
LIN {X 0,Y 473.815,Z 749.345,A -85,B 0,C 180,E1 7867.71,E2 7867.71} C_VEL
LIN {X 0,Y 473.341,Z 736.712,A -85,B 0,C 180,E1 7867.997,E2 7867.997} C_VEL
LIN {X 0,Y 449.89,Z 689.128,A -85,B 0,C 180,E1 7871.024,E2 7871.024} C_VEL
LIN {X 0,Y 448.753,Z 685.03,A -85,B 0,C 180,E1 7871.296,E2 7871.296} C_VEL
LIN {X 0,Y 448.66,Z 685.03,A -85,B 0,C 180,E1 7877.726,E2 7877.726} C_VEL
LIN {X 0,Y 448.819,Z 685.03,A -85,B 0,C 180,E1 7883.795,E2 7883.795} C_VEL
LIN {X 0,Y 448.808,Z 685.03,A -85,B 0,C 180,E1 7889.711,E2 7889.711} C_VEL
LIN {X 0,Y 448.84,Z 685.03,A -85,B 0,C 180,E1 7896.205,E2 7896.205} C_VEL
LIN {X 0,Y 449.103,Z 685.03,A -85,B 0,C 180,E1 7902.396,E2 7902.396} C_VEL
LIN {X 0,Y 449.263,Z 685.03,A -85,B 0,C 180,E1 7908.371,E2 7908.371} C_VEL
LIN {X 0,Y 449.51,Z 685.03,A -85,B 0,C 180,E1 7914.217,E2 7914.217} C_VEL
LIN {X 0,Y 449.702,Z 685.03,A -85,B 0,C 180,E1 7919.996,E2 7919.996} C_VEL
LIN {X 0,Y 449.53,Z 685.03,A -85,B 0,C 180,E1 7925.776,E2 7925.776} C_VEL
LIN {X 0,Y 449.267,Z 685.03,A -85,B 0,C 180,E1 7931.622,E2 7931.622} C_VEL
LIN {X 0,Y 449.094,Z 685.03,A -85,B 0,C 180,E1 7937.597,E2 7937.597} C_VEL
LIN {X 0,Y 448.919,Z 685.03,A -85,B 0,C 180,E1 7943.783,E2 7943.783} C_VEL
LIN {X 0,Y 448.683,Z 685.03,A -85,B 0,C 180,E1 7950.29,E2 7950.29} C_VEL
LIN {X 0,Y 448.731,Z 685.03,A -85,B 0,C 180,E1 7957.243,E2 7957.243} C_VEL
LIN {X 0,Y 448.694,Z 685.03,A -85,B 0,C 180,E1 7962.279,E2 7962.279} C_VEL
LIN {X 0,Y 448.616,Z 685.03,A -85,B 0,C 180,E1 7967.722,E2 7967.722} C_VEL
LIN {X 0,Y 448.661,Z 685.03,A -85,B 0,C 180,E1 7973.811,E2 7973.811} C_VEL
LIN {X 0,Y 448.757,Z 685.662,A -85,B 0,C 180,E1 7975.309,E2 7975.309} C_VEL
LIN {X 0,Y 462.765,Z 718.375,A -85,B 0,C 180,E1 7978.552,E2 7978.552} C_VEL
LIN {X 0,Y 467.212,Z 735.823,A -85,B 0,C 180,E1 7980.292,E2 7980.292} C_VEL
LIN {X 0,Y 463.311,Z 765.82,A -85,B 0,C 180,E1 7982.872,E2 7982.872} C_VEL
LIN {X 0,Y 459.337,Z 792.391,A -85,B 0,C 180,E1 7986.012,E2 7986.012} C_VEL
LIN {X 0,Y 455.474,Z 816.481,A -85,B 0,C 180,E1 7989.896,E2 7989.896} C_VEL
LIN {X 0,Y 452.765,Z 835.111,A -85,B 0,C 180,E1 7994.04,E2 7994.04} C_VEL
LIN {X 0,Y 451.019,Z 850.223,A -85,B 0,C 180,E1 7998.908,E2 7998.908} C_VEL
LIN {X 0,Y 450.368,Z 858.73,A -85,B 0,C 180,E1 8003.265,E2 8003.265} C_VEL
LIN {X 0,Y 450.151,Z 863.176,A -85,B 0,C 180,E1 8008.079,E2 8008.079} C_VEL
LIN {X 0,Y 450.203,Z 863.122,A -85,B 0,C 180,E1 8011.921,E2 8011.921} C_VEL
LIN {X 0,Y 450.345,Z 858.601,A -85,B 0,C 180,E1 8016.735,E2 8016.735} C_VEL
LIN {X 0,Y 451.158,Z 848.793,A -85,B 0,C 180,E1 8021.577,E2 8021.577} C_VEL
LIN {X 0,Y 453.099,Z 832.815,A -85,B 0,C 180,E1 8026.444,E2 8026.444} C_VEL
LIN {X 0,Y 455.964,Z 813.343,A -85,B 0,C 180,E1 8030.587,E2 8030.587} C_VEL
LIN {X 0,Y 459.901,Z 788.247,A -85,B 0,C 180,E1 8034.472,E2 8034.472} C_VEL
LIN {X 0,Y 464.229,Z 758.811,A -85,B 0,C 180,E1 8037.725,E2 8037.725} C_VEL
LIN {X 0,Y 466.965,Z 732.533,A -85,B 0,C 180,E1 8039.917,E2 8039.917} C_VEL
LIN {X 0,Y 459.058,Z 709.314,A -85,B 0,C 180,E1 8042.304,E2 8042.304} C_VEL
LIN {X 0,Y 448.703,Z 685.03,A -85,B 0,C 180,E1 8044.679,E2 8044.679} C_VEL
LIN {X 0,Y 448.651,Z 685.03,A -85,B 0,C 180,E1 8049.721,E2 8049.721} C_VEL
LIN {X 0,Y 448.65,Z 685.03,A -85,B 0,C 180,E1 8055.073,E2 8055.073} C_VEL
LIN {X 0,Y 448.747,Z 685.03,A -85,B 0,C 180,E1 8060.662,E2 8060.662} C_VEL
LIN {X 0,Y 448.682,Z 685.03,A -85,B 0,C 180,E1 8067.452,E2 8067.452} C_VEL
LIN {X 0,Y 448.901,Z 685.03,A -85,B 0,C 180,E1 8074.094,E2 8074.094} C_VEL
LIN {X 0,Y 449.101,Z 685.03,A -85,B 0,C 180,E1 8080.372,E2 8080.372} C_VEL
LIN {X 0,Y 449.376,Z 685.03,A -85,B 0,C 180,E1 8086.858,E2 8086.858} C_VEL
LIN {X 0,Y 449.403,Z 685.03,A -85,B 0,C 180,E1 8092.665,E2 8092.665} C_VEL
LIN {X 0,Y 449.601,Z 685.03,A -85,B 0,C 180,E1 8098.08,E2 8098.08} C_VEL
LIN {X 0,Y 449.569,Z 685.03,A -85,B 0,C 180,E1 8103.853,E2 8103.853} C_VEL
LIN {X 0,Y 449.311,Z 685.03,A -85,B 0,C 180,E1 8109.67,E2 8109.67} C_VEL
LIN {X 0,Y 449.138,Z 685.03,A -85,B 0,C 180,E1 8115.594,E2 8115.594} C_VEL
LIN {X 0,Y 448.965,Z 685.03,A -85,B 0,C 180,E1 8121.7,E2 8121.7} C_VEL
LIN {X 0,Y 448.764,Z 685.03,A -85,B 0,C 180,E1 8128.085,E2 8128.085} C_VEL
LIN {X 0,Y 448.573,Z 685.03,A -85,B 0,C 180,E1 8134.883,E2 8134.883} C_VEL
LIN {X 0,Y 448.578,Z 685.03,A -85,B 0,C 180,E1 8139.73,E2 8139.73} C_VEL
LIN {X 0,Y 448.574,Z 685.03,A -85,B 0,C 180,E1 8145.055,E2 8145.055} C_VEL
LIN {X 0,Y 448.753,Z 685.03,A -85,B 0,C 180,E1 8148.767,E2 8148.767} C_VEL
LIN {X 0,Y 455.164,Z 698.941,A -85,B 0,C 180,E1 8149.687,E2 8149.687} C_VEL
LIN {X 0,Y 473.959,Z 738.894,A -85,B 0,C 180,E1 8152.092,E2 8152.092} C_VEL
LIN {X 0,Y 472.006,Z 783.566,A -85,B 0,C 180,E1 8153.153,E2 8153.153} C_VEL
LIN {X 0,Y 468.772,Z 823.675,A -85,B 0,C 180,E1 8154.843,E2 8154.843} C_VEL
LIN {X 0,Y 467.253,Z 839.531,A -85,B 0,C 180,E1 8155.736,E2 8155.736} C_VEL
LIN {X 0,Y 461.853,Z 855.029,A -85,B 0,C 180,E1 8156.523,E2 8156.523} C_VEL
LIN {X 0,Y 457.047,Z 868.099,A -85,B 0,C 180,E1 8157.32,E2 8157.32} C_VEL
LIN {X 0,Y 456.777,Z 869.92,A -85,B 0,C 180,E1 8157.467,E2 8157.467} C_VEL
LIN {X 0,Y 452.481,Z 905.475,A -85,B 0,C 180,E1 8160.808,E2 8160.808} C_VEL
LIN {X 0,Y 448.741,Z 936.021,A -85,B 0,C 180,E1 8164.635,E2 8164.635} C_VEL
LIN {X 0,Y 445.801,Z 961.007,A -85,B 0,C 180,E1 8168.72,E2 8168.72} C_VEL
LIN {X 0,Y 443.9,Z 979.399,A -85,B 0,C 180,E1 8172.696,E2 8172.696} C_VEL
LIN {X 0,Y 442.569,Z 995.067,A -85,B 0,C 180,E1 8177.696,E2 8177.696} C_VEL
LIN {X 0,Y 442.092,Z 1004.218,A -85,B 0,C 180,E1 8182.153,E2 8182.153} C_VEL
LIN {X 0,Y 441.907,Z 1008.907,A -85,B 0,C 180,E1 8186.084,E2 8186.084} C_VEL
LIN {X 0,Y 441.953,Z 1010.5,A -85,B 0,C 180,E1 8190,E2 8190} C_VEL
LIN {X 0,Y 441.896,Z 1008.91,A -85,B 0,C 180,E1 8193.916,E2 8193.916} C_VEL
LIN {X 0,Y 442.19,Z 1002.518,A -85,B 0,C 180,E1 8198.874,E2 8198.874} C_VEL
LIN {X 0,Y 442.921,Z 991.04,A -85,B 0,C 180,E1 8203.797,E2 8203.797} C_VEL
LIN {X 0,Y 444.454,Z 974.297,A -85,B 0,C 180,E1 8208.564,E2 8208.564} C_VEL
LIN {X 0,Y 447.029,Z 950.704,A -85,B 0,C 180,E1 8213.105,E2 8213.105} C_VEL
LIN {X 0,Y 450.615,Z 920.669,A -85,B 0,C 180,E1 8217.418,E2 8217.418} C_VEL
LIN {X 0,Y 454.492,Z 889.021,A -85,B 0,C 180,E1 8220.857,E2 8220.857} C_VEL
LIN {X 0,Y 458.676,Z 853.295,A -85,B 0,C 180,E1 8223.773,E2 8223.773} C_VEL
LIN {X 0,Y 462.377,Z 816.262,A -85,B 0,C 180,E1 8225.976,E2 8225.976} C_VEL
LIN {X 0,Y 465.695,Z 777.062,A -85,B 0,C 180,E1 8227.532,E2 8227.532} C_VEL
LIN {X 0,Y 466.871,Z 739.757,A -85,B 0,C 180,E1 8228.464,E2 8228.464} C_VEL
LIN {X 0,Y 443.058,Z 690.559,A -85,B 0,C 180,E1 8231.677,E2 8231.677} C_VEL
LIN {X 0,Y 440.796,Z 685.03,A -85,B 0,C 180,E1 8232.104,E2 8232.104} C_VEL
LIN {X 0,Y 440.722,Z 685.03,A -85,B 0,C 180,E1 8239.416,E2 8239.416} C_VEL
LIN {X 0,Y 440.907,Z 685.03,A -85,B 0,C 180,E1 8245.224,E2 8245.224} C_VEL
LIN {X 0,Y 440.889,Z 685.03,A -85,B 0,C 180,E1 8251.367,E2 8251.367} C_VEL
LIN {X 0,Y 440.974,Z 685.03,A -85,B 0,C 180,E1 8257.886,E2 8257.886} C_VEL
LIN {X 0,Y 441.264,Z 685.03,A -85,B 0,C 180,E1 8264.12,E2 8264.12} C_VEL
LIN {X 0,Y 441.448,Z 685.03,A -85,B 0,C 180,E1 8270.156,E2 8270.156} C_VEL
LIN {X 0,Y 441.734,Z 685.03,A -85,B 0,C 180,E1 8276.079,E2 8276.079} C_VEL
LIN {X 0,Y 441.895,Z 685.03,A -85,B 0,C 180,E1 8281.953,E2 8281.953} C_VEL
LIN {X 0,Y 441.529,Z 685.03,A -85,B 0,C 180,E1 8287.853,E2 8287.853} C_VEL
LIN {X 0,Y 441.326,Z 685.03,A -85,B 0,C 180,E1 8293.843,E2 8293.843} C_VEL
LIN {X 0,Y 441.117,Z 685.03,A -85,B 0,C 180,E1 8299.998,E2 8299.998} C_VEL
LIN {X 0,Y 440.889,Z 685.03,A -85,B 0,C 180,E1 8306.413,E2 8306.413} C_VEL
LIN {X 0,Y 440.695,Z 685.03,A -85,B 0,C 180,E1 8313.213,E2 8313.213} C_VEL
LIN {X 0,Y 440.788,Z 685.03,A -85,B 0,C 180,E1 8318.059,E2 8318.059} C_VEL
LIN {X 0,Y 440.652,Z 685.03,A -85,B 0,C 180,E1 8324.017,E2 8324.017} C_VEL
LIN {X 0,Y 440.63,Z 685.03,A -85,B 0,C 180,E1 8329.407,E2 8329.407} C_VEL
LIN {X 0,Y 440.782,Z 685.342,A -85,B 0,C 180,E1 8334.444,E2 8334.444} C_VEL
LIN {X 0,Y 454.595,Z 717.424,A -85,B 0,C 180,E1 8337.69,E2 8337.69} C_VEL
LIN {X 0,Y 460.539,Z 737.625,A -85,B 0,C 180,E1 8339.818,E2 8339.818} C_VEL
LIN {X 0,Y 456.474,Z 767.508,A -85,B 0,C 180,E1 8342.432,E2 8342.432} C_VEL
LIN {X 0,Y 452.274,Z 794.067,A -85,B 0,C 180,E1 8345.614,E2 8345.614} C_VEL
LIN {X 0,Y 448.209,Z 818.173,A -85,B 0,C 180,E1 8349.556,E2 8349.556} C_VEL
LIN {X 0,Y 445.293,Z 836.647,A -85,B 0,C 180,E1 8353.765,E2 8353.765} C_VEL
LIN {X 0,Y 443.454,Z 850.44,A -85,B 0,C 180,E1 8358.219,E2 8358.219} C_VEL
LIN {X 0,Y 442.614,Z 860.074,A -85,B 0,C 180,E1 8363.147,E2 8363.147} C_VEL
LIN {X 0,Y 442.391,Z 864.485,A -85,B 0,C 180,E1 8368.045,E2 8368.045} C_VEL
LIN {X 0,Y 442.442,Z 864.432,A -85,B 0,C 180,E1 8371.955,E2 8371.955} C_VEL
LIN {X 0,Y 442.595,Z 859.946,A -85,B 0,C 180,E1 8376.853,E2 8376.853} C_VEL
LIN {X 0,Y 443.536,Z 850.213,A -85,B 0,C 180,E1 8381.779,E2 8381.779} C_VEL
LIN {X 0,Y 445.635,Z 834.387,A -85,B 0,C 180,E1 8386.728,E2 8386.728} C_VEL
LIN {X 0,Y 448.733,Z 815.029,A -85,B 0,C 180,E1 8390.934,E2 8390.934} C_VEL
LIN {X 0,Y 452.571,Z 791.69,A -85,B 0,C 180,E1 8394.632,E2 8394.632} C_VEL
LIN {X 0,Y 457.157,Z 762.532,A -85,B 0,C 180,E1 8397.989,E2 8397.989} C_VEL
LIN {X 0,Y 460.345,Z 735.77,A -85,B 0,C 180,E1 8400.269,E2 8400.269} C_VEL
LIN {X 0,Y 452.178,Z 711.741,A -85,B 0,C 180,E1 8402.834,E2 8402.834} C_VEL
LIN {X 0,Y 440.759,Z 685.03,A -85,B 0,C 180,E1 8405.592,E2 8405.592} C_VEL
LIN {X 0,Y 440.663,Z 685.03,A -85,B 0,C 180,E1 8411.128,E2 8411.128} C_VEL
LIN {X 0,Y 440.696,Z 685.03,A -85,B 0,C 180,E1 8416.787,E2 8416.787} C_VEL
LIN {X 0,Y 440.79,Z 685.03,A -85,B 0,C 180,E1 8421.968,E2 8421.968} C_VEL
LIN {X 0,Y 440.737,Z 685.03,A -85,B 0,C 180,E1 8426.791,E2 8426.791} C_VEL
LIN {X 0,Y 440.92,Z 685.03,A -85,B 0,C 180,E1 8433.589,E2 8433.589} C_VEL
LIN {X 0,Y 441.17,Z 685.03,A -85,B 0,C 180,E1 8440.004,E2 8440.004} C_VEL
LIN {X 0,Y 441.438,Z 685.03,A -85,B 0,C 180,E1 8446.161,E2 8446.161} C_VEL
LIN {X 0,Y 441.528,Z 685.03,A -85,B 0,C 180,E1 8452.658,E2 8452.658} C_VEL
LIN {X 0,Y 441.697,Z 685.03,A -85,B 0,C 180,E1 8458.046,E2 8458.046} C_VEL
LIN {X 0,Y 441.659,Z 685.03,A -85,B 0,C 180,E1 8463.922,E2 8463.922} C_VEL
LIN {X 0,Y 441.398,Z 685.03,A -85,B 0,C 180,E1 8469.845,E2 8469.845} C_VEL
LIN {X 0,Y 441.197,Z 685.03,A -85,B 0,C 180,E1 8475.882,E2 8475.882} C_VEL
LIN {X 0,Y 440.963,Z 685.03,A -85,B 0,C 180,E1 8482.489,E2 8482.489} C_VEL
LIN {X 0,Y 440.841,Z 685.03,A -85,B 0,C 180,E1 8488.636,E2 8488.636} C_VEL
LIN {X 0,Y 440.662,Z 685.03,A -85,B 0,C 180,E1 8495.603,E2 8495.603} C_VEL
LIN {X 0,Y 440.565,Z 685.03,A -85,B 0,C 180,E1 8501.103,E2 8501.103} C_VEL
LIN {X 0,Y 440.78,Z 685.03,A -85,B 0,C 180,E1 8507.966,E2 8507.966} C_VEL
LIN {X 0,Y 445.41,Z 695.204,A -85,B 0,C 180,E1 8508.663,E2 8508.663} C_VEL
LIN {X 0,Y 467.19,Z 740.356,A -85,B 0,C 180,E1 8511.574,E2 8511.574} C_VEL
LIN {X 0,Y 465.106,Z 784.208,A -85,B 0,C 180,E1 8512.691,E2 8512.691} C_VEL
LIN {X 0,Y 461.63,Z 824.2,A -85,B 0,C 180,E1 8514.432,E2 8514.432} C_VEL
LIN {X 0,Y 457.665,Z 861.645,A -85,B 0,C 180,E1 8516.828,E2 8516.828} C_VEL
LIN {X 0,Y 456.777,Z 869.92,A -85,B 0,C 180,E1 8517.467,E2 8517.467} C_VEL
LIN {X 0,Y 454.772,Z 877.298,A -85,B 0,C 180,E1 8518.032,E2 8518.032} C_VEL
LIN {X 0,Y 446.08,Z 896.442,A -85,B 0,C 180,E1 8519.55,E2 8519.55} C_VEL
LIN {X 0,Y 445.8,Z 898.115,A -85,B 0,C 180,E1 8519.72,E2 8519.72} C_VEL
LIN {X 0,Y 441.679,Z 930.492,A -85,B 0,C 180,E1 8523.631,E2 8523.631} C_VEL
LIN {X 0,Y 438.243,Z 958.53,A -85,B 0,C 180,E1 8528.165,E2 8528.165} C_VEL
LIN {X 0,Y 435.932,Z 980.205,A -85,B 0,C 180,E1 8532.889,E2 8532.889} C_VEL
LIN {X 0,Y 434.705,Z 995.256,A -85,B 0,C 180,E1 8537.544,E2 8537.544} C_VEL
LIN {X 0,Y 434.218,Z 1004.218,A -85,B 0,C 180,E1 8542.01,E2 8542.01} C_VEL
LIN {X 0,Y 434.025,Z 1008.906,A -85,B 0,C 180,E1 8546.013,E2 8546.013} C_VEL
LIN {X 0,Y 434.053,Z 1010.5,A -85,B 0,C 180,E1 8550,E2 8550} C_VEL
LIN {X 0,Y 434.016,Z 1008.91,A -85,B 0,C 180,E1 8553.987,E2 8553.987} C_VEL
LIN {X 0,Y 434.297,Z 1002.598,A -85,B 0,C 180,E1 8558.995,E2 8558.995} C_VEL
LIN {X 0,Y 435.1,Z 990.887,A -85,B 0,C 180,E1 8564.05,E2 8564.05} C_VEL
LIN {X 0,Y 436.685,Z 972.777,A -85,B 0,C 180,E1 8568.902,E2 8568.902} C_VEL
LIN {X 0,Y 439.404,Z 948.988,A -85,B 0,C 180,E1 8573.53,E2 8573.53} C_VEL
LIN {X 0,Y 443.124,Z 919.503,A -85,B 0,C 180,E1 8577.819,E2 8577.819} C_VEL
LIN {X 0,Y 447.235,Z 886.972,A -85,B 0,C 180,E1 8581.391,E2 8581.391} C_VEL
LIN {X 0,Y 451.65,Z 850.924,A -85,B 0,C 180,E1 8584.352,E2 8584.352} C_VEL
LIN {X 0,Y 455.828,Z 811.888,A -85,B 0,C 180,E1 8586.666,E2 8586.666} C_VEL
LIN {X 0,Y 459.209,Z 773.914,A -85,B 0,C 180,E1 8588.157,E2 8588.157} C_VEL
LIN {X 0,Y 460.2,Z 742.28,A -85,B 0,C 180,E1 8588.982,E2 8588.982} C_VEL
LIN {X 0,Y 437.706,Z 695.481,A -85,B 0,C 180,E1 8592.125,E2 8592.125} C_VEL
LIN {X 0,Y 432.765,Z 685.03,A -85,B 0,C 180,E1 8592.924,E2 8592.924} C_VEL
LIN {X 0,Y 432.769,Z 685.03,A -85,B 0,C 180,E1 8600.094,E2 8600.094} C_VEL
LIN {X 0,Y 433.003,Z 685.03,A -85,B 0,C 180,E1 8606.76,E2 8606.76} C_VEL
LIN {X 0,Y 432.957,Z 685.03,A -85,B 0,C 180,E1 8613.056,E2 8613.056} C_VEL
LIN {X 0,Y 433.179,Z 685.03,A -85,B 0,C 180,E1 8620.145,E2 8620.145} C_VEL
LIN {X 0,Y 433.409,Z 685.03,A -85,B 0,C 180,E1 8625.891,E2 8625.891} C_VEL
LIN {X 0,Y 433.572,Z 685.03,A -85,B 0,C 180,E1 8631.994,E2 8631.994} C_VEL
LIN {X 0,Y 433.812,Z 685.03,A -85,B 0,C 180,E1 8638.003,E2 8638.003} C_VEL
LIN {X 0,Y 433.75,Z 685.03,A -85,B 0,C 180,E1 8643.986,E2 8643.986} C_VEL
LIN {X 0,Y 433.486,Z 685.03,A -85,B 0,C 180,E1 8650.019,E2 8650.019} C_VEL
LIN {X 0,Y 433.322,Z 685.03,A -85,B 0,C 180,E1 8656.171,E2 8656.171} C_VEL
LIN {X 0,Y 433.114,Z 685.03,A -85,B 0,C 180,E1 8662.529,E2 8662.529} C_VEL
LIN {X 0,Y 432.821,Z 685.03,A -85,B 0,C 180,E1 8669.355,E2 8669.355} C_VEL
LIN {X 0,Y 432.787,Z 685.03,A -85,B 0,C 180,E1 8676.344,E2 8676.344} C_VEL
LIN {X 0,Y 432.787,Z 685.03,A -85,B 0,C 180,E1 8682.929,E2 8682.929} C_VEL
LIN {X 0,Y 432.663,Z 685.03,A -85,B 0,C 180,E1 8690.1,E2 8690.1} C_VEL
LIN {X 0,Y 432.777,Z 685.141,A -85,B 0,C 180,E1 8693.542,E2 8693.542} C_VEL
LIN {X 0,Y 447.407,Z 719.186,A -85,B 0,C 180,E1 8697.089,E2 8697.089} C_VEL
LIN {X 0,Y 453.733,Z 739.399,A -85,B 0,C 180,E1 8699.317,E2 8699.317} C_VEL
LIN {X 0,Y 449.41,Z 770.562,A -85,B 0,C 180,E1 8702.124,E2 8702.124} C_VEL
LIN {X 0,Y 444.585,Z 799.134,A -85,B 0,C 180,E1 8705.698,E2 8705.698} C_VEL
LIN {X 0,Y 440.462,Z 822.176,A -85,B 0,C 180,E1 8709.704,E2 8709.704} C_VEL
LIN {X 0,Y 437.533,Z 839.932,A -85,B 0,C 180,E1 8713.984,E2 8713.984} C_VEL
LIN {X 0,Y 435.625,Z 854.253,A -85,B 0,C 180,E1 8719.017,E2 8719.017} C_VEL
LIN {X 0,Y 434.824,Z 862.716,A -85,B 0,C 180,E1 8724.024,E2 8724.024} C_VEL
LIN {X 0,Y 434.628,Z 865.796,A -85,B 0,C 180,E1 8728.01,E2 8728.01} C_VEL
LIN {X 0,Y 434.671,Z 865.746,A -85,B 0,C 180,E1 8731.989,E2 8731.989} C_VEL
LIN {X 0,Y 434.869,Z 861.304,A -85,B 0,C 180,E1 8736.976,E2 8736.976} C_VEL
LIN {X 0,Y 435.9,Z 851.654,A -85,B 0,C 180,E1 8741.988,E2 8741.988} C_VEL
LIN {X 0,Y 438.185,Z 835.943,A -85,B 0,C 180,E1 8747.021,E2 8747.021} C_VEL
LIN {X 0,Y 441.502,Z 816.582,A -85,B 0,C 180,E1 8751.294,E2 8751.294} C_VEL
LIN {X 0,Y 445.534,Z 793.26,A -85,B 0,C 180,E1 8755.047,E2 8755.047} C_VEL
LIN {X 0,Y 450.267,Z 764.783,A -85,B 0,C 180,E1 8758.388,E2 8758.388} C_VEL
LIN {X 0,Y 453.474,Z 737.574,A -85,B 0,C 180,E1 8760.777,E2 8760.777} C_VEL
LIN {X 0,Y 444.411,Z 711.864,A -85,B 0,C 180,E1 8763.622,E2 8763.622} C_VEL
LIN {X 0,Y 432.757,Z 685.03,A -85,B 0,C 180,E1 8766.439,E2 8766.439} C_VEL
LIN {X 0,Y 432.756,Z 685.03,A -85,B 0,C 180,E1 8772.934,E2 8772.934} C_VEL
LIN {X 0,Y 432.782,Z 685.03,A -85,B 0,C 180,E1 8778.52,E2 8778.52} C_VEL
LIN {X 0,Y 432.806,Z 685.03,A -85,B 0,C 180,E1 8783.658,E2 8783.658} C_VEL
LIN {X 0,Y 432.794,Z 685.03,A -85,B 0,C 180,E1 8788.474,E2 8788.474} C_VEL
LIN {X 0,Y 433.028,Z 685.03,A -85,B 0,C 180,E1 8795.287,E2 8795.287} C_VEL
LIN {X 0,Y 433.294,Z 685.03,A -85,B 0,C 180,E1 8801.739,E2 8801.739} C_VEL
LIN {X 0,Y 433.543,Z 685.03,A -85,B 0,C 180,E1 8807.951,E2 8807.951} C_VEL
LIN {X 0,Y 433.694,Z 685.03,A -85,B 0,C 180,E1 8814.013,E2 8814.013} C_VEL
LIN {X 0,Y 433.9,Z 685.03,A -85,B 0,C 180,E1 8820.004,E2 8820.004} C_VEL
LIN {X 0,Y 433.708,Z 685.03,A -85,B 0,C 180,E1 8825.995,E2 8825.995} C_VEL
LIN {X 0,Y 433.363,Z 685.03,A -85,B 0,C 180,E1 8832.845,E2 8832.845} C_VEL
LIN {X 0,Y 433.217,Z 685.03,A -85,B 0,C 180,E1 8838.272,E2 8838.272} C_VEL
LIN {X 0,Y 432.951,Z 685.03,A -85,B 0,C 180,E1 8845.015,E2 8845.015} C_VEL
LIN {X 0,Y 432.723,Z 685.03,A -85,B 0,C 180,E1 8851.541,E2 8851.541} C_VEL
LIN {X 0,Y 432.653,Z 685.03,A -85,B 0,C 180,E1 8856.661,E2 8856.661} C_VEL
LIN {X 0,Y 432.626,Z 685.03,A -85,B 0,C 180,E1 8862.906,E2 8862.906} C_VEL
LIN {X 0,Y 432.787,Z 685.103,A -85,B 0,C 180,E1 8867.123,E2 8867.123} C_VEL
LIN {X 0,Y 437.368,Z 695.044,A -85,B 0,C 180,E1 8867.834,E2 8867.834} C_VEL
LIN {X 0,Y 454.98,Z 731.174,A -85,B 0,C 180,E1 8870.324,E2 8870.324} C_VEL
LIN {X 0,Y 460.682,Z 744.38,A -85,B 0,C 180,E1 8871.108,E2 8871.108} C_VEL
LIN {X 0,Y 458.243,Z 785.852,A -85,B 0,C 180,E1 8872.235,E2 8872.235} C_VEL
LIN {X 0,Y 454.564,Z 824.57,A -85,B 0,C 180,E1 8873.997,E2 8873.997} C_VEL
LIN {X 0,Y 450.201,Z 863.04,A -85,B 0,C 180,E1 8876.542,E2 8876.542} C_VEL
LIN {X 0,Y 445.8,Z 898.115,A -85,B 0,C 180,E1 8879.72,E2 8879.72} C_VEL
LIN {X 0,Y 443.792,Z 904.859,A -85,B 0,C 180,E1 8880.395,E2 8880.395} C_VEL
LIN {X 0,Y 435.128,Z 922.273,A -85,B 0,C 180,E1 8882.284,E2 8882.284} C_VEL
LIN {X 0,Y 434.857,Z 923.779,A -85,B 0,C 180,E1 8882.488,E2 8882.488} C_VEL
LIN {X 0,Y 431.263,Z 951.736,A -85,B 0,C 180,E1 8886.819,E2 8886.819} C_VEL
LIN {X 0,Y 428.631,Z 974.473,A -85,B 0,C 180,E1 8891.528,E2 8891.528} C_VEL
LIN {X 0,Y 427.147,Z 990.958,A -85,B 0,C 180,E1 8896.18,E2 8896.18} C_VEL
LIN {X 0,Y 426.436,Z 1002.318,A -85,B 0,C 180,E1 8900.837,E2 8900.837} C_VEL
LIN {X 0,Y 426.192,Z 1006.928,A -85,B 0,C 180,E1 8903.903,E2 8903.903} C_VEL
LIN {X 0,Y 426.125,Z 1010.089,A -85,B 0,C 180,E1 8907.971,E2 8907.971} C_VEL
LIN {X 0,Y 426.164,Z 1010.09,A -85,B 0,C 180,E1 8912.029,E2 8912.029} C_VEL
LIN {X 0,Y 426.327,Z 1004.836,A -85,B 0,C 180,E1 8917.667,E2 8917.667} C_VEL
LIN {X 0,Y 426.942,Z 994.305,A -85,B 0,C 180,E1 8922.647,E2 8922.647} C_VEL
LIN {X 0,Y 428.387,Z 977.953,A -85,B 0,C 180,E1 8927.623,E2 8927.623} C_VEL
LIN {X 0,Y 430.857,Z 954.619,A -85,B 0,C 180,E1 8932.659,E2 8932.659} C_VEL
LIN {X 0,Y 434.347,Z 927.451,A -85,B 0,C 180,E1 8937.007,E2 8937.007} C_VEL
LIN {X 0,Y 438.676,Z 895.351,A -85,B 0,C 180,E1 8940.891,E2 8940.891} C_VEL
LIN {X 0,Y 443.345,Z 860.346,A -85,B 0,C 180,E1 8944.072,E2 8944.072} C_VEL
LIN {X 0,Y 447.841,Z 822.794,A -85,B 0,C 180,E1 8946.595,E2 8946.595} C_VEL
LIN {X 0,Y 451.723,Z 784.409,A -85,B 0,C 180,E1 8948.356,E2 8948.356} C_VEL
LIN {X 0,Y 453.749,Z 745.015,A -85,B 0,C 180,E1 8949.492,E2 8949.492} C_VEL
LIN {X 0,Y 432.522,Z 700.463,A -85,B 0,C 180,E1 8952.568,E2 8952.568} C_VEL
LIN {X 0,Y 424.893,Z 686.247,A -85,B 0,C 180,E1 8953.741,E2 8953.741} C_VEL
LIN {X 0,Y 424.809,Z 685.03,A -85,B 0,C 180,E1 8953.931,E2 8953.931} C_VEL
LIN {X 0,Y 424.871,Z 685.03,A -85,B 0,C 180,E1 8960.259,E2 8960.259} C_VEL
LIN {X 0,Y 424.973,Z 685.03,A -85,B 0,C 180,E1 8965.378,E2 8965.378} C_VEL
LIN {X 0,Y 424.981,Z 685.03,A -85,B 0,C 180,E1 8970.189,E2 8970.189} C_VEL
LIN {X 0,Y 425.133,Z 685.03,A -85,B 0,C 180,E1 8977.348,E2 8977.348} C_VEL
LIN {X 0,Y 425.383,Z 685.03,A -85,B 0,C 180,E1 8983.511,E2 8983.511} C_VEL
LIN {X 0,Y 425.584,Z 685.03,A -85,B 0,C 180,E1 8989.785,E2 8989.785} C_VEL
LIN {X 0,Y 425.904,Z 685.03,A -85,B 0,C 180,E1 8995.933,E2 8995.933} C_VEL
LIN {X 0,Y 426.071,Z 685.03,A -85,B 0,C 180,E1 9002.026,E2 9002.026} C_VEL
LIN {X 0,Y 425.674,Z 685.03,A -85,B 0,C 180,E1 9008.147,E2 9008.147} C_VEL
LIN {X 0,Y 425.451,Z 685.03,A -85,B 0,C 180,E1 9014.37,E2 9014.37} C_VEL
LIN {X 0,Y 425.229,Z 685.03,A -85,B 0,C 180,E1 9020.779,E2 9020.779} C_VEL
LIN {X 0,Y 424.976,Z 685.03,A -85,B 0,C 180,E1 9027.484,E2 9027.484} C_VEL
LIN {X 0,Y 424.81,Z 685.03,A -85,B 0,C 180,E1 9034.627,E2 9034.627} C_VEL
LIN {X 0,Y 424.853,Z 685.03,A -85,B 0,C 180,E1 9039.733,E2 9039.733} C_VEL
LIN {X 0,Y 424.812,Z 685.03,A -85,B 0,C 180,E1 9045.26,E2 9045.26} C_VEL
LIN {X 0,Y 424.802,Z 685.03,A -85,B 0,C 180,E1 9052.577,E2 9052.577} C_VEL
LIN {X 0,Y 439.77,Z 719.562,A -85,B 0,C 180,E1 9056.314,E2 9056.314} C_VEL
LIN {X 0,Y 446.891,Z 741.247,A -85,B 0,C 180,E1 9058.804,E2 9058.804} C_VEL
LIN {X 0,Y 442.51,Z 772.746,A -85,B 0,C 180,E1 9061.721,E2 9061.721} C_VEL
LIN {X 0,Y 437.524,Z 800.63,A -85,B 0,C 180,E1 9065.28,E2 9065.28} C_VEL
LIN {X 0,Y 433.165,Z 823.644,A -85,B 0,C 180,E1 9069.346,E2 9069.346} C_VEL
LIN {X 0,Y 429.888,Z 842.412,A -85,B 0,C 180,E1 9073.997,E2 9073.997} C_VEL
LIN {X 0,Y 427.962,Z 855.676,A -85,B 0,C 180,E1 9078.818,E2 9078.818} C_VEL
LIN {X 0,Y 427.067,Z 864.06,A -85,B 0,C 180,E1 9083.915,E2 9083.915} C_VEL
LIN {X 0,Y 426.867,Z 867.106,A -85,B 0,C 180,E1 9087.974,E2 9087.974} C_VEL
LIN {X 0,Y 426.909,Z 867.058,A -85,B 0,C 180,E1 9092.026,E2 9092.026} C_VEL
LIN {X 0,Y 427.126,Z 862.66,A -85,B 0,C 180,E1 9097.103,E2 9097.103} C_VEL
LIN {X 0,Y 428.285,Z 853.078,A -85,B 0,C 180,E1 9102.204,E2 9102.204} C_VEL
LIN {X 0,Y 430.726,Z 837.411,A -85,B 0,C 180,E1 9107.325,E2 9107.325} C_VEL
LIN {X 0,Y 434.252,Z 818.068,A -85,B 0,C 180,E1 9111.667,E2 9111.667} C_VEL
LIN {X 0,Y 438.512,Z 794.784,A -85,B 0,C 180,E1 9115.477,E2 9115.477} C_VEL
LIN {X 0,Y 443.543,Z 766.038,A -85,B 0,C 180,E1 9118.897,E2 9118.897} C_VEL
LIN {X 0,Y 446.668,Z 739.667,A -85,B 0,C 180,E1 9121.267,E2 9121.267} C_VEL
LIN {X 0,Y 436.698,Z 712.176,A -85,B 0,C 180,E1 9124.425,E2 9124.425} C_VEL
LIN {X 0,Y 424.824,Z 685.03,A -85,B 0,C 180,E1 9127.321,E2 9127.321} C_VEL
LIN {X 0,Y 424.828,Z 685.03,A -85,B 0,C 180,E1 9132.445,E2 9132.445} C_VEL
LIN {X 0,Y 424.873,Z 685.03,A -85,B 0,C 180,E1 9138.231,E2 9138.231} C_VEL
LIN {X 0,Y 424.848,Z 685.03,A -85,B 0,C 180,E1 9144.778,E2 9144.778} C_VEL
LIN {X 0,Y 424.909,Z 685.03,A -85,B 0,C 180,E1 9150.193,E2 9150.193} C_VEL
LIN {X 0,Y 425.208,Z 685.03,A -85,B 0,C 180,E1 9157.323,E2 9157.323} C_VEL
LIN {X 0,Y 425.468,Z 685.03,A -85,B 0,C 180,E1 9163.522,E2 9163.522} C_VEL
LIN {X 0,Y 425.64,Z 685.03,A -85,B 0,C 180,E1 9169.794,E2 9169.794} C_VEL
LIN {X 0,Y 425.878,Z 685.03,A -85,B 0,C 180,E1 9175.941,E2 9175.941} C_VEL
LIN {X 0,Y 426.074,Z 685.03,A -85,B 0,C 180,E1 9182.033,E2 9182.033} C_VEL
LIN {X 0,Y 425.675,Z 685.03,A -85,B 0,C 180,E1 9188.155,E2 9188.155} C_VEL
LIN {X 0,Y 425.42,Z 685.03,A -85,B 0,C 180,E1 9194.38,E2 9194.38} C_VEL
LIN {X 0,Y 425.185,Z 685.03,A -85,B 0,C 180,E1 9200.79,E2 9200.79} C_VEL
LIN {X 0,Y 424.989,Z 685.03,A -85,B 0,C 180,E1 9207.492,E2 9207.492} C_VEL
LIN {X 0,Y 424.817,Z 685.03,A -85,B 0,C 180,E1 9212.198,E2 9212.198} C_VEL
LIN {X 0,Y 424.686,Z 685.03,A -85,B 0,C 180,E1 9218.583,E2 9218.583} C_VEL
LIN {X 0,Y 424.744,Z 685.03,A -85,B 0,C 180,E1 9225.28,E2 9225.28} C_VEL
LIN {X 0,Y 424.793,Z 685.03,A -85,B 0,C 180,E1 9226.22,E2 9226.22} C_VEL
LIN {X 0,Y 427.25,Z 690.726,A -85,B 0,C 180,E1 9226.636,E2 9226.636} C_VEL
LIN {X 0,Y 446.423,Z 728.937,A -85,B 0,C 180,E1 9229.473,E2 9229.473} C_VEL
LIN {X 0,Y 454.101,Z 747.418,A -85,B 0,C 180,E1 9230.598,E2 9230.598} C_VEL
LIN {X 0,Y 451.428,Z 787.688,A -85,B 0,C 180,E1 9231.764,E2 9231.764} C_VEL
LIN {X 0,Y 447.469,Z 826.151,A -85,B 0,C 180,E1 9233.595,E2 9233.595} C_VEL
LIN {X 0,Y 442.759,Z 864.46,A -85,B 0,C 180,E1 9236.247,E2 9236.247} C_VEL
LIN {X 0,Y 437.78,Z 901.95,A -85,B 0,C 180,E1 9239.815,E2 9239.815} C_VEL
LIN {X 0,Y 434.857,Z 923.779,A -85,B 0,C 180,E1 9242.488,E2 9242.488} C_VEL
LIN {X 0,Y 431.264,Z 932.765,A -85,B 0,C 180,E1 9243.68,E2 9243.68} C_VEL
LIN {X 0,Y 424.332,Z 945.148,A -85,B 0,C 180,E1 9245.525,E2 9245.525} C_VEL
LIN {X 0,Y 424.071,Z 946.51,A -85,B 0,C 180,E1 9245.753,E2 9245.753} C_VEL
LIN {X 0,Y 421.18,Z 970.779,A -85,B 0,C 180,E1 9250.646,E2 9250.646} C_VEL
LIN {X 0,Y 419.322,Z 989.728,A -85,B 0,C 180,E1 9255.994,E2 9255.994} C_VEL
LIN {X 0,Y 418.612,Z 1000.956,A -85,B 0,C 180,E1 9260.665,E2 9260.665} C_VEL
LIN {X 0,Y 418.276,Z 1008.007,A -85,B 0,C 180,E1 9265.862,E2 9265.862} C_VEL
LIN {X 0,Y 418.283,Z 1009.791,A -85,B 0,C 180,E1 9270,E2 9270} C_VEL
LIN {X 0,Y 418.258,Z 1007.044,A -85,B 0,C 180,E1 9275.175,E2 9275.175} C_VEL
LIN {X 0,Y 418.619,Z 999.883,A -85,B 0,C 180,E1 9279.859,E2 9279.859} C_VEL
LIN {X 0,Y 419.452,Z 988.029,A -85,B 0,C 180,E1 9284.586,E2 9284.586} C_VEL
LIN {X 0,Y 421.2,Z 969.619,A -85,B 0,C 180,E1 9289.625,E2 9289.625} C_VEL
LIN {X 0,Y 424.158,Z 945.46,A -85,B 0,C 180,E1 9294.423,E2 9294.423} C_VEL
LIN {X 0,Y 428.13,Z 916.589,A -85,B 0,C 180,E1 9298.724,E2 9298.724} C_VEL
LIN {X 0,Y 433.007,Z 882.236,A -85,B 0,C 180,E1 9302.581,E2 9302.581} C_VEL
LIN {X 0,Y 438.141,Z 845.132,A -85,B 0,C 180,E1 9305.686,E2 9305.686} C_VEL
LIN {X 0,Y 443.05,Z 804.983,A -85,B 0,C 180,E1 9308.054,E2 9308.054} C_VEL
LIN {X 0,Y 447.051,Z 762.829,A -85,B 0,C 180,E1 9309.601,E2 9309.601} C_VEL
LIN {X 0,Y 447.18,Z 747.533,A -85,B 0,C 180,E1 9310.038,E2 9310.038} C_VEL
LIN {X 0,Y 427.356,Z 705.407,A -85,B 0,C 180,E1 9313.024,E2 9313.024} C_VEL
LIN {X 0,Y 416.891,Z 685.638,A -85,B 0,C 180,E1 9314.701,E2 9314.701} C_VEL
LIN {X 0,Y 417.014,Z 685.03,A -85,B 0,C 180,E1 9322.035,E2 9322.035} C_VEL
LIN {X 0,Y 417.025,Z 685.03,A -85,B 0,C 180,E1 9327.126,E2 9327.126} C_VEL
LIN {X 0,Y 417.03,Z 685.03,A -85,B 0,C 180,E1 9331.938,E2 9331.938} C_VEL
LIN {X 0,Y 417.25,Z 685.03,A -85,B 0,C 180,E1 9338.796,E2 9338.796} C_VEL
LIN {X 0,Y 417.542,Z 685.03,A -85,B 0,C 180,E1 9345.343,E2 9345.343} C_VEL
LIN {X 0,Y 417.728,Z 685.03,A -85,B 0,C 180,E1 9351.689,E2 9351.689} C_VEL
LIN {X 0,Y 418.034,Z 685.03,A -85,B 0,C 180,E1 9357.928,E2 9357.928} C_VEL
LIN {X 0,Y 417.926,Z 685.03,A -85,B 0,C 180,E1 9364.137,E2 9364.137} C_VEL
LIN {X 0,Y 417.63,Z 685.03,A -85,B 0,C 180,E1 9370.403,E2 9370.403} C_VEL
LIN {X 0,Y 417.441,Z 685.03,A -85,B 0,C 180,E1 9376.804,E2 9376.804} C_VEL
LIN {X 0,Y 417.191,Z 685.03,A -85,B 0,C 180,E1 9383.439,E2 9383.439} C_VEL
LIN {X 0,Y 416.951,Z 685.03,A -85,B 0,C 180,E1 9390.436,E2 9390.436} C_VEL
LIN {X 0,Y 416.961,Z 685.03,A -85,B 0,C 180,E1 9397.961,E2 9397.961} C_VEL
LIN {X 0,Y 416.862,Z 685.03,A -85,B 0,C 180,E1 9403.616,E2 9403.616} C_VEL
LIN {X 0,Y 416.806,Z 685.03,A -85,B 0,C 180,E1 9409.478,E2 9409.478} C_VEL
LIN {X 0,Y 416.899,Z 685.262,A -85,B 0,C 180,E1 9411.661,E2 9411.661} C_VEL
LIN {X 0,Y 429.363,Z 713.054,A -85,B 0,C 180,E1 9414.719,E2 9414.719} C_VEL
LIN {X 0,Y 439.503,Z 740.667,A -85,B 0,C 180,E1 9417.993,E2 9417.993} C_VEL
LIN {X 0,Y 439.807,Z 748.942,A -85,B 0,C 180,E1 9418.803,E2 9418.803} C_VEL
LIN {X 0,Y 434.929,Z 778.494,A -85,B 0,C 180,E1 9421.713,E2 9421.713} C_VEL
LIN {X 0,Y 429.884,Z 804.966,A -85,B 0,C 180,E1 9425.298,E2 9425.298} C_VEL
LIN {X 0,Y 425.446,Z 827.322,A -85,B 0,C 180,E1 9429.456,E2 9429.456} C_VEL
LIN {X 0,Y 422.043,Z 846.185,A -85,B 0,C 180,E1 9434.453,E2 9434.453} C_VEL
LIN {X 0,Y 420.091,Z 859.098,A -85,B 0,C 180,E1 9439.653,E2 9439.653} C_VEL
LIN {X 0,Y 419.305,Z 865.399,A -85,B 0,C 180,E1 9443.802,E2 9443.802} C_VEL
LIN {X 0,Y 419.101,Z 868.419,A -85,B 0,C 180,E1 9447.937,E2 9447.937} C_VEL
LIN {X 0,Y 419.138,Z 868.371,A -85,B 0,C 180,E1 9452.063,E2 9452.063} C_VEL
LIN {X 0,Y 419.415,Z 864.005,A -85,B 0,C 180,E1 9457.234,E2 9457.234} C_VEL
LIN {X 0,Y 420.646,Z 854.463,A -85,B 0,C 180,E1 9462.43,E2 9462.43} C_VEL
LIN {X 0,Y 423.284,Z 838.831,A -85,B 0,C 180,E1 9467.639,E2 9467.639} C_VEL
LIN {X 0,Y 427.318,Z 818.173,A -85,B 0,C 180,E1 9472.31,E2 9472.31} C_VEL
LIN {X 0,Y 431.908,Z 794.48,A -85,B 0,C 180,E1 9476.173,E2 9476.173} C_VEL
LIN {X 0,Y 437.281,Z 764.648,A -85,B 0,C 180,E1 9479.681,E2 9479.681} C_VEL
LIN {X 0,Y 440.212,Z 743.594,A -85,B 0,C 180,E1 9481.569,E2 9481.569} C_VEL
LIN {X 0,Y 430.163,Z 715.042,A -85,B 0,C 180,E1 9484.96,E2 9484.96} C_VEL
LIN {X 0,Y 416.931,Z 685.636,A -85,B 0,C 180,E1 9488.22,E2 9488.22} C_VEL
LIN {X 0,Y 416.855,Z 685.03,A -85,B 0,C 180,E1 9493.625,E2 9493.625} C_VEL
LIN {X 0,Y 416.914,Z 685.03,A -85,B 0,C 180,E1 9499.471,E2 9499.471} C_VEL
LIN {X 0,Y 416.934,Z 685.03,A -85,B 0,C 180,E1 9504.622,E2 9504.622} C_VEL
LIN {X 0,Y 417.028,Z 685.03,A -85,B 0,C 180,E1 9511.947,E2 9511.947} C_VEL
LIN {X 0,Y 417.327,Z 685.03,A -85,B 0,C 180,E1 9518.808,E2 9518.808} C_VEL
LIN {X 0,Y 417.643,Z 685.03,A -85,B 0,C 180,E1 9525.355,E2 9525.355} C_VEL
LIN {X 0,Y 417.762,Z 685.03,A -85,B 0,C 180,E1 9531.697,E2 9531.697} C_VEL
LIN {X 0,Y 417.983,Z 685.03,A -85,B 0,C 180,E1 9537.935,E2 9537.935} C_VEL
LIN {X 0,Y 417.928,Z 685.03,A -85,B 0,C 180,E1 9544.145,E2 9544.145} C_VEL
LIN {X 0,Y 417.614,Z 685.03,A -85,B 0,C 180,E1 9550.412,E2 9550.412} C_VEL
LIN {X 0,Y 417.411,Z 685.03,A -85,B 0,C 180,E1 9556.814,E2 9556.814} C_VEL
LIN {X 0,Y 417.135,Z 685.03,A -85,B 0,C 180,E1 9563.451,E2 9563.451} C_VEL
LIN {X 0,Y 416.91,Z 685.03,A -85,B 0,C 180,E1 9570.448,E2 9570.448} C_VEL
LIN {X 0,Y 416.797,Z 685.03,A -85,B 0,C 180,E1 9577.203,E2 9577.203} C_VEL
LIN {X 0,Y 416.749,Z 685.03,A -85,B 0,C 180,E1 9583.6,E2 9583.6} C_VEL
LIN {X 0,Y 416.864,Z 685.232,A -85,B 0,C 180,E1 9585.293,E2 9585.293} C_VEL
LIN {X 0,Y 421.609,Z 695.201,A -85,B 0,C 180,E1 9586.092,E2 9586.092} C_VEL
LIN {X 0,Y 439.338,Z 729.91,A -85,B 0,C 180,E1 9588.793,E2 9588.793} C_VEL
LIN {X 0,Y 447.595,Z 748.479,A -85,B 0,C 180,E1 9590.025,E2 9590.025} C_VEL
LIN {X 0,Y 444.455,Z 791.729,A -85,B 0,C 180,E1 9591.362,E2 9591.362} C_VEL
LIN {X 0,Y 439.929,Z 831.807,A -85,B 0,C 180,E1 9593.428,E2 9593.428} C_VEL
LIN {X 0,Y 435.013,Z 868.327,A -85,B 0,C 180,E1 9596.139,E2 9596.139} C_VEL
LIN {X 0,Y 429.948,Z 903.985,A -85,B 0,C 180,E1 9599.733,E2 9599.733} C_VEL
LIN {X 0,Y 425.786,Z 933.849,A -85,B 0,C 180,E1 9603.704,E2 9603.704} C_VEL
LIN {X 0,Y 424.071,Z 946.51,A -85,B 0,C 180,E1 9605.753,E2 9605.753} C_VEL
LIN {X 0,Y 422.147,Z 951.778,A -85,B 0,C 180,E1 9606.663,E2 9606.663} C_VEL
LIN {X 0,Y 413.941,Z 964.698,A -85,B 0,C 180,E1 9609.247,E2 9609.247} C_VEL
LIN {X 0,Y 413.735,Z 965.837,A -85,B 0,C 180,E1 9609.505,E2 9609.505} C_VEL
LIN {X 0,Y 411.8,Z 984.867,A -85,B 0,C 180,E1 9614.593,E2 9614.593} C_VEL
LIN {X 0,Y 410.908,Z 998.525,A -85,B 0,C 180,E1 9619.954,E2 9619.954} C_VEL
LIN {X 0,Y 410.45,Z 1005.709,A -85,B 0,C 180,E1 9624.726,E2 9624.726} C_VEL
LIN {X 0,Y 410.499,Z 1008.481,A -85,B 0,C 180,E1 9630,E2 9630} C_VEL
LIN {X 0,Y 410.466,Z 1005.714,A -85,B 0,C 180,E1 9635.273,E2 9635.273} C_VEL
LIN {X 0,Y 410.822,Z 998.502,A -85,B 0,C 180,E1 9640.048,E2 9640.048} C_VEL
LIN {X 0,Y 411.636,Z 986.559,A -85,B 0,C 180,E1 9644.869,E2 9644.869} C_VEL
LIN {X 0,Y 413.504,Z 967.986,A -85,B 0,C 180,E1 9650.006,E2 9650.006} C_VEL
LIN {X 0,Y 416.509,Z 944.483,A -85,B 0,C 180,E1 9654.753,E2 9654.753} C_VEL
LIN {X 0,Y 420.651,Z 915.492,A -85,B 0,C 180,E1 9659.157,E2 9659.157} C_VEL
LIN {X 0,Y 425.691,Z 882.254,A -85,B 0,C 180,E1 9663.001,E2 9663.001} C_VEL
LIN {X 0,Y 430.944,Z 846.798,A -85,B 0,C 180,E1 9666.065,E2 9666.065} C_VEL
LIN {X 0,Y 435.961,Z 808.185,A -85,B 0,C 180,E1 9668.451,E2 9668.451} C_VEL
LIN {X 0,Y 440.042,Z 769.534,A -85,B 0,C 180,E1 9670,E2 9670} C_VEL
LIN {X 0,Y 440.725,Z 750.117,A -85,B 0,C 180,E1 9670.595,E2 9670.595} C_VEL
LIN {X 0,Y 422.009,Z 709.923,A -85,B 0,C 180,E1 9673.526,E2 9673.526} C_VEL
LIN {X 0,Y 409.111,Z 686.697,A -85,B 0,C 180,E1 9675.645,E2 9675.645} C_VEL
LIN {X 0,Y 408.938,Z 685.03,A -85,B 0,C 180,E1 9675.76,E2 9675.76} C_VEL
LIN {X 0,Y 408.987,Z 685.03,A -85,B 0,C 180,E1 9681.152,E2 9681.152} C_VEL
LIN {X 0,Y 409.122,Z 685.03,A -85,B 0,C 180,E1 9686.407,E2 9686.407} C_VEL
LIN {X 0,Y 409.088,Z 685.03,A -85,B 0,C 180,E1 9693.725,E2 9693.725} C_VEL
LIN {X 0,Y 409.387,Z 685.03,A -85,B 0,C 180,E1 9700.623,E2 9700.623} C_VEL
LIN {X 0,Y 409.698,Z 685.03,A -85,B 0,C 180,E1 9707.23,E2 9707.23} C_VEL
LIN {X 0,Y 409.937,Z 685.03,A -85,B 0,C 180,E1 9713.656,E2 9713.656} C_VEL
LIN {X 0,Y 410.207,Z 685.03,A -85,B 0,C 180,E1 9719.996,E2 9719.996} C_VEL
LIN {X 0,Y 409.95,Z 685.03,A -85,B 0,C 180,E1 9726.36,E2 9726.36} C_VEL
LIN {X 0,Y 409.705,Z 685.03,A -85,B 0,C 180,E1 9732.762,E2 9732.762} C_VEL
LIN {X 0,Y 409.415,Z 685.03,A -85,B 0,C 180,E1 9739.367,E2 9739.367} C_VEL
LIN {X 0,Y 409.115,Z 685.03,A -85,B 0,C 180,E1 9746.264,E2 9746.264} C_VEL
LIN {X 0,Y 408.961,Z 685.03,A -85,B 0,C 180,E1 9753.598,E2 9753.598} C_VEL
LIN {X 0,Y 408.934,Z 685.03,A -85,B 0,C 180,E1 9759.203,E2 9759.203} C_VEL
LIN {X 0,Y 408.826,Z 685.03,A -85,B 0,C 180,E1 9765.469,E2 9765.469} C_VEL
LIN {X 0,Y 408.908,Z 685.466,A -85,B 0,C 180,E1 9770.644,E2 9770.644} C_VEL
LIN {X 0,Y 424.19,Z 719.261,A -85,B 0,C 180,E1 9774.546,E2 9774.546} C_VEL
LIN {X 0,Y 433.285,Z 745.42,A -85,B 0,C 180,E1 9777.778,E2 9777.778} C_VEL
LIN {X 0,Y 428.679,Z 777.158,A -85,B 0,C 180,E1 9780.885,E2 9780.885} C_VEL
LIN {X 0,Y 423.089,Z 805.18,A -85,B 0,C 180,E1 9784.66,E2 9784.66} C_VEL
LIN {X 0,Y 418.356,Z 827.708,A -85,B 0,C 180,E1 9788.857,E2 9788.857} C_VEL
LIN {X 0,Y 414.761,Z 845.941,A -85,B 0,C 180,E1 9793.623,E2 9793.623} C_VEL
LIN {X 0,Y 412.522,Z 859.438,A -85,B 0,C 180,E1 9798.928,E2 9798.928} C_VEL
LIN {X 0,Y 411.554,Z 866.726,A -85,B 0,C 180,E1 9803.685,E2 9803.685} C_VEL
LIN {X 0,Y 411.34,Z 869.728,A -85,B 0,C 180,E1 9807.898,E2 9807.898} C_VEL
LIN {X 0,Y 411.375,Z 869.682,A -85,B 0,C 180,E1 9812.102,E2 9812.102} C_VEL
LIN {X 0,Y 411.691,Z 865.337,A -85,B 0,C 180,E1 9817.371,E2 9817.371} C_VEL
LIN {X 0,Y 413.033,Z 855.822,A -85,B 0,C 180,E1 9822.662,E2 9822.662} C_VEL
LIN {X 0,Y 415.841,Z 840.232,A -85,B 0,C 180,E1 9827.966,E2 9827.966} C_VEL
LIN {X 0,Y 419.829,Z 820.947,A -85,B 0,C 180,E1 9832.451,E2 9832.451} C_VEL
LIN {X 0,Y 424.578,Z 797.743,A -85,B 0,C 180,E1 9836.376,E2 9836.376} C_VEL
LIN {X 0,Y 430.004,Z 769.435,A -85,B 0,C 180,E1 9839.861,E2 9839.861} C_VEL
LIN {X 0,Y 433.641,Z 746.782,A -85,B 0,C 180,E1 9841.961,E2 9841.961} C_VEL
LIN {X 0,Y 423.659,Z 717.944,A -85,B 0,C 180,E1 9845.508,E2 9845.508} C_VEL
LIN {X 0,Y 409.02,Z 685.71,A -85,B 0,C 180,E1 9849.229,E2 9849.229} C_VEL
LIN {X 0,Y 408.871,Z 685.03,A -85,B 0,C 180,E1 9855.485,E2 9855.485} C_VEL
LIN {X 0,Y 408.955,Z 685.03,A -85,B 0,C 180,E1 9861.159,E2 9861.159} C_VEL
LIN {X 0,Y 408.997,Z 685.03,A -85,B 0,C 180,E1 9866.405,E2 9866.405} C_VEL
LIN {X 0,Y 409.162,Z 685.03,A -85,B 0,C 180,E1 9873.739,E2 9873.739} C_VEL
LIN {X 0,Y 409.473,Z 685.03,A -85,B 0,C 180,E1 9880.636,E2 9880.636} C_VEL
LIN {X 0,Y 409.798,Z 685.03,A -85,B 0,C 180,E1 9887.241,E2 9887.241} C_VEL
LIN {X 0,Y 409.954,Z 685.03,A -85,B 0,C 180,E1 9893.665,E2 9893.665} C_VEL
LIN {X 0,Y 410.207,Z 685.03,A -85,B 0,C 180,E1 9900.004,E2 9900.004} C_VEL
LIN {X 0,Y 409.957,Z 685.03,A -85,B 0,C 180,E1 9906.368,E2 9906.368} C_VEL
LIN {X 0,Y 409.659,Z 685.03,A -85,B 0,C 180,E1 9912.772,E2 9912.772} C_VEL
LIN {X 0,Y 409.387,Z 685.03,A -85,B 0,C 180,E1 9919.377,E2 9919.377} C_VEL
LIN {X 0,Y 409.087,Z 685.03,A -85,B 0,C 180,E1 9926.275,E2 9926.275} C_VEL
LIN {X 0,Y 408.909,Z 685.03,A -85,B 0,C 180,E1 9933.612,E2 9933.612} C_VEL
LIN {X 0,Y 408.766,Z 685.03,A -85,B 0,C 180,E1 9939.174,E2 9939.174} C_VEL
LIN {X 0,Y 408.926,Z 685.397,A -85,B 0,C 180,E1 9944.308,E2 9944.308} C_VEL
LIN {X 0,Y 414.191,Z 695.886,A -85,B 0,C 180,E1 9945.223,E2 9945.223} C_VEL
LIN {X 0,Y 433.213,Z 732.722,A -85,B 0,C 180,E1 9948.223,E2 9948.223} C_VEL
LIN {X 0,Y 441.134,Z 752.463,A -85,B 0,C 180,E1 9949.519,E2 9949.519} C_VEL
LIN {X 0,Y 437.657,Z 793.492,A -85,B 0,C 180,E1 9950.869,E2 9950.869} C_VEL
LIN {X 0,Y 433.096,Z 831.72,A -85,B 0,C 180,E1 9952.902,E2 9952.902} C_VEL
LIN {X 0,Y 427.902,Z 867.942,A -85,B 0,C 180,E1 9955.651,E2 9955.651} C_VEL
LIN {X 0,Y 422.675,Z 902.421,A -85,B 0,C 180,E1 9959.205,E2 9959.205} C_VEL
LIN {X 0,Y 418.054,Z 933.708,A -85,B 0,C 180,E1 9963.469,E2 9963.469} C_VEL
LIN {X 0,Y 414.427,Z 960.101,A -85,B 0,C 180,E1 9968.244,E2 9968.244} C_VEL
LIN {X 0,Y 413.735,Z 965.837,A -85,B 0,C 180,E1 9969.505,E2 9969.505} C_VEL
LIN {X 0,Y 412.043,Z 970.216,A -85,B 0,C 180,E1 9970.532,E2 9970.532} C_VEL
LIN {X 0,Y 404.315,Z 980.651,A -85,B 0,C 180,E1 9973.419,E2 9973.419} C_VEL
LIN {X 0,Y 404.134,Z 981.531,A -85,B 0,C 180,E1 9973.702,E2 9973.702} C_VEL
LIN {X 0,Y 403.152,Z 994.942,A -85,B 0,C 180,E1 9978.667,E2 9978.667} C_VEL
LIN {X 0,Y 402.76,Z 1003.149,A -85,B 0,C 180,E1 9983.546,E2 9983.546} C_VEL
LIN {X 0,Y 402.663,Z 1006.696,A -85,B 0,C 180,E1 9987.852,E2 9987.852} C_VEL
LIN {X 0,Y 402.698,Z 1006.702,A -85,B 0,C 180,E1 9992.147,E2 9992.147} C_VEL
LIN {X 0,Y 402.824,Z 1002.095,A -85,B 0,C 180,E1 9997.295,E2 9997.295} C_VEL
LIN {X 0,Y 403.332,Z 992.386,A -85,B 0,C 180,E1 10002.423,E2 10002.423} C_VEL
LIN {X 0,Y 404.598,Z 977.953,A -85,B 0,C 180,E1 10007.36,E2 10007.36} C_VEL
LIN {X 0,Y 406.908,Z 957.571,A -85,B 0,C 180,E1 10012.356,E2 10012.356} C_VEL
LIN {X 0,Y 410.61,Z 931.862,A -85,B 0,C 180,E1 10017.051,E2 10017.051} C_VEL
LIN {X 0,Y 415.593,Z 900.295,A -85,B 0,C 180,E1 10021.43,E2 10021.43} C_VEL
LIN {X 0,Y 421.065,Z 866.163,A -85,B 0,C 180,E1 10024.988,E2 10024.988} C_VEL
LIN {X 0,Y 426.817,Z 827.841,A -85,B 0,C 180,E1 10027.9,E2 10027.9} C_VEL
LIN {X 0,Y 431.853,Z 787.123,A -85,B 0,C 180,E1 10029.99,E2 10029.99} C_VEL
LIN {X 0,Y 434.429,Z 753.205,A -85,B 0,C 180,E1 10031.117,E2 10031.117} C_VEL
LIN {X 0,Y 416.91,Z 714.777,A -85,B 0,C 180,E1 10034.007,E2 10034.007} C_VEL
LIN {X 0,Y 401.1,Z 686.235,A -85,B 0,C 180,E1 10036.712,E2 10036.712} C_VEL
LIN {X 0,Y 400.991,Z 685.03,A -85,B 0,C 180,E1 10036.953,E2 10036.953} C_VEL
LIN {X 0,Y 401.069,Z 685.03,A -85,B 0,C 180,E1 10042.986,E2 10042.986} C_VEL
LIN {X 0,Y 401.189,Z 685.03,A -85,B 0,C 180,E1 10048.223,E2 10048.223} C_VEL
LIN {X 0,Y 401.209,Z 685.03,A -85,B 0,C 180,E1 10055.558,E2 10055.558} C_VEL
LIN {X 0,Y 401.554,Z 685.03,A -85,B 0,C 180,E1 10062.502,E2 10062.502} C_VEL
LIN {X 0,Y 401.816,Z 685.03,A -85,B 0,C 180,E1 10069.174,E2 10069.174} C_VEL
LIN {X 0,Y 402.171,Z 685.03,A -85,B 0,C 180,E1 10075.693,E2 10075.693} C_VEL
LIN {X 0,Y 402.381,Z 685.03,A -85,B 0,C 180,E1 10082.145,E2 10082.145} C_VEL
LIN {X 0,Y 401.886,Z 685.03,A -85,B 0,C 180,E1 10088.633,E2 10088.633} C_VEL
LIN {X 0,Y 401.669,Z 685.03,A -85,B 0,C 180,E1 10095.241,E2 10095.241} C_VEL
LIN {X 0,Y 401.39,Z 685.03,A -85,B 0,C 180,E1 10102.076,E2 10102.076} C_VEL
LIN {X 0,Y 401.049,Z 685.03,A -85,B 0,C 180,E1 10109.277,E2 10109.277} C_VEL
LIN {X 0,Y 401.018,Z 685.03,A -85,B 0,C 180,E1 10114.355,E2 10114.355} C_VEL
LIN {X 0,Y 400.942,Z 685.03,A -85,B 0,C 180,E1 10121.173,E2 10121.173} C_VEL
LIN {X 0,Y 400.892,Z 685.03,A -85,B 0,C 180,E1 10127.349,E2 10127.349} C_VEL
LIN {X 0,Y 400.982,Z 685.275,A -85,B 0,C 180,E1 10129.56,E2 10129.56} C_VEL
LIN {X 0,Y 409.662,Z 703.909,A -85,B 0,C 180,E1 10131.734,E2 10131.734} C_VEL
LIN {X 0,Y 421.732,Z 733.133,A -85,B 0,C 180,E1 10135.369,E2 10135.369} C_VEL
LIN {X 0,Y 426.88,Z 750.767,A -85,B 0,C 180,E1 10137.607,E2 10137.607} C_VEL
LIN {X 0,Y 421.43,Z 780.992,A -85,B 0,C 180,E1 10140.653,E2 10140.653} C_VEL
LIN {X 0,Y 415.79,Z 807.934,A -85,B 0,C 180,E1 10144.416,E2 10144.416} C_VEL
LIN {X 0,Y 410.794,Z 830.499,A -85,B 0,C 180,E1 10148.772,E2 10148.772} C_VEL
LIN {X 0,Y 407.241,Z 847.489,A -85,B 0,C 180,E1 10153.367,E2 10153.367} C_VEL
LIN {X 0,Y 404.837,Z 860.783,A -85,B 0,C 180,E1 10158.715,E2 10158.715} C_VEL
LIN {X 0,Y 403.795,Z 868.05,A -85,B 0,C 180,E1 10163.563,E2 10163.563} C_VEL
LIN {X 0,Y 403.551,Z 871.042,A -85,B 0,C 180,E1 10167.857,E2 10167.857} C_VEL
LIN {X 0,Y 403.586,Z 870.996,A -85,B 0,C 180,E1 10172.143,E2 10172.143} C_VEL
LIN {X 0,Y 403.913,Z 866.918,A -85,B 0,C 180,E1 10177.317,E2 10177.317} C_VEL
LIN {X 0,Y 405.399,Z 857.177,A -85,B 0,C 180,E1 10182.905,E2 10182.905} C_VEL
LIN {X 0,Y 408.414,Z 841.618,A -85,B 0,C 180,E1 10188.304,E2 10188.304} C_VEL
LIN {X 0,Y 412.635,Z 822.364,A -85,B 0,C 180,E1 10192.864,E2 10192.864} C_VEL
LIN {X 0,Y 417.644,Z 799.2,A -85,B 0,C 180,E1 10196.849,E2 10196.849} C_VEL
LIN {X 0,Y 423.207,Z 771.475,A -85,B 0,C 180,E1 10200.327,E2 10200.327} C_VEL
LIN {X 0,Y 426.851,Z 749.151,A -85,B 0,C 180,E1 10202.468,E2 10202.468} C_VEL
LIN {X 0,Y 416.244,Z 718.563,A -85,B 0,C 180,E1 10206.349,E2 10206.349} C_VEL
LIN {X 0,Y 402.297,Z 689.28,A -85,B 0,C 180,E1 10209.969,E2 10209.969} C_VEL
LIN {X 0,Y 401.063,Z 685.03,A -85,B 0,C 180,E1 10210.365,E2 10210.365} C_VEL
LIN {X 0,Y 400.964,Z 685.03,A -85,B 0,C 180,E1 10217.368,E2 10217.368} C_VEL
LIN {X 0,Y 401.004,Z 685.03,A -85,B 0,C 180,E1 10222.989,E2 10222.989} C_VEL
LIN {X 0,Y 401.06,Z 685.03,A -85,B 0,C 180,E1 10229.926,E2 10229.926} C_VEL
LIN {X 0,Y 401.283,Z 685.03,A -85,B 0,C 180,E1 10235.572,E2 10235.572} C_VEL
LIN {X 0,Y 401.618,Z 685.03,A -85,B 0,C 180,E1 10242.513,E2 10242.513} C_VEL
LIN {X 0,Y 401.883,Z 685.03,A -85,B 0,C 180,E1 10249.184,E2 10249.184} C_VEL
LIN {X 0,Y 402.152,Z 685.03,A -85,B 0,C 180,E1 10255.701,E2 10255.701} C_VEL
LIN {X 0,Y 402.384,Z 685.03,A -85,B 0,C 180,E1 10262.153,E2 10262.153} C_VEL
LIN {X 0,Y 401.884,Z 685.03,A -85,B 0,C 180,E1 10268.642,E2 10268.642} C_VEL
LIN {X 0,Y 401.628,Z 685.03,A -85,B 0,C 180,E1 10275.251,E2 10275.251} C_VEL
LIN {X 0,Y 401.345,Z 685.03,A -85,B 0,C 180,E1 10282.088,E2 10282.088} C_VEL
LIN {X 0,Y 401.041,Z 685.03,A -85,B 0,C 180,E1 10289.287,E2 10289.287} C_VEL
LIN {X 0,Y 400.962,Z 685.03,A -85,B 0,C 180,E1 10294.371,E2 10294.371} C_VEL
LIN {X 0,Y 400.81,Z 685.03,A -85,B 0,C 180,E1 10301.152,E2 10301.152} C_VEL
LIN {X 0,Y 400.93,Z 685.03,A -85,B 0,C 180,E1 10303.241,E2 10303.241} C_VEL
LIN {X 0,Y 403.488,Z 690.816,A -85,B 0,C 180,E1 10303.735,E2 10303.735} C_VEL
LIN {X 0,Y 425.013,Z 730.947,A -85,B 0,C 180,E1 10307.301,E2 10307.301} C_VEL
LIN {X 0,Y 434.62,Z 754.83,A -85,B 0,C 180,E1 10308.958,E2 10308.958} C_VEL
LIN {X 0,Y 430.951,Z 794.947,A -85,B 0,C 180,E1 10310.346,E2 10310.346} C_VEL
LIN {X 0,Y 426.253,Z 831.774,A -85,B 0,C 180,E1 10312.362,E2 10312.362} C_VEL
LIN {X 0,Y 420.856,Z 867.408,A -85,B 0,C 180,E1 10315.126,E2 10315.126} C_VEL
LIN {X 0,Y 415.335,Z 901.645,A -85,B 0,C 180,E1 10318.732,E2 10318.732} C_VEL
LIN {X 0,Y 410.605,Z 931.867,A -85,B 0,C 180,E1 10322.949,E2 10322.949} C_VEL
LIN {X 0,Y 406.869,Z 957.659,A -85,B 0,C 180,E1 10327.658,E2 10327.658} C_VEL
LIN {X 0,Y 404.475,Z 977.945,A -85,B 0,C 180,E1 10332.635,E2 10332.635} C_VEL
LIN {X 0,Y 404.134,Z 981.531,A -85,B 0,C 180,E1 10333.702,E2 10333.702} C_VEL
LIN {X 0,Y 401.194,Z 986.448,A -85,B 0,C 180,E1 10335.387,E2 10335.387} C_VEL
LIN {X 0,Y 395.494,Z 992.489,A -85,B 0,C 180,E1 10337.986,E2 10337.986} C_VEL
LIN {X 0,Y 395.371,Z 993.17,A -85,B 0,C 180,E1 10338.288,E2 10338.288} C_VEL
LIN {X 0,Y 394.963,Z 1001.805,A -85,B 0,C 180,E1 10343.418,E2 10343.418} C_VEL
LIN {X 0,Y 394.874,Z 1005.38,A -85,B 0,C 180,E1 10347.81,E2 10347.81} C_VEL
LIN {X 0,Y 394.908,Z 1005.387,A -85,B 0,C 180,E1 10352.19,E2 10352.19} C_VEL
LIN {X 0,Y 395.031,Z 1000.579,A -85,B 0,C 180,E1 10357.573,E2 10357.573} C_VEL
LIN {X 0,Y 395.61,Z 989.651,A -85,B 0,C 180,E1 10363.23,E2 10363.23} C_VEL
LIN {X 0,Y 397.026,Z 973.884,A -85,B 0,C 180,E1 10368.437,E2 10368.437} C_VEL
LIN {X 0,Y 400.085,Z 950.576,A -85,B 0,C 180,E1 10373.92,E2 10373.92} C_VEL
LIN {X 0,Y 404.521,Z 922.2,A -85,B 0,C 180,E1 10378.844,E2 10378.844} C_VEL
LIN {X 0,Y 409.843,Z 890.555,A -85,B 0,C 180,E1 10382.991,E2 10382.991} C_VEL
LIN {X 0,Y 415.675,Z 855.964,A -85,B 0,C 180,E1 10386.382,E2 10386.382} C_VEL
LIN {X 0,Y 421.239,Z 819.42,A -85,B 0,C 180,E1 10388.986,E2 10388.986} C_VEL
LIN {X 0,Y 426.038,Z 781.906,A -85,B 0,C 180,E1 10390.8,E2 10390.8} C_VEL
LIN {X 0,Y 427.926,Z 755.612,A -85,B 0,C 180,E1 10391.701,E2 10391.701} C_VEL
LIN {X 0,Y 412.028,Z 720.056,A -85,B 0,C 180,E1 10394.468,E2 10394.468} C_VEL
LIN {X 0,Y 393.136,Z 686.214,A -85,B 0,C 180,E1 10397.826,E2 10397.826} C_VEL
LIN {X 0,Y 393.018,Z 685.03,A -85,B 0,C 180,E1 10397.992,E2 10397.992} C_VEL
LIN {X 0,Y 393.154,Z 685.03,A -85,B 0,C 180,E1 10404.847,E2 10404.847} C_VEL
LIN {X 0,Y 393.19,Z 685.03,A -85,B 0,C 180,E1 10411.97,E2 10411.97} C_VEL
LIN {X 0,Y 393.353,Z 685.03,A -85,B 0,C 180,E1 10417.439,E2 10417.439} C_VEL
LIN {X 0,Y 393.726,Z 685.03,A -85,B 0,C 180,E1 10424.435,E2 10424.435} C_VEL
LIN {X 0,Y 393.964,Z 685.03,A -85,B 0,C 180,E1 10431.183,E2 10431.183} C_VEL
LIN {X 0,Y 394.327,Z 685.03,A -85,B 0,C 180,E1 10437.803,E2 10437.803} C_VEL
LIN {X 0,Y 394.206,Z 685.03,A -85,B 0,C 180,E1 10444.386,E2 10444.386} C_VEL
LIN {X 0,Y 393.876,Z 685.03,A -85,B 0,C 180,E1 10451.039,E2 10451.039} C_VEL
LIN {X 0,Y 393.605,Z 685.03,A -85,B 0,C 180,E1 10457.855,E2 10457.855} C_VEL
LIN {X 0,Y 393.317,Z 685.03,A -85,B 0,C 180,E1 10464.956,E2 10464.956} C_VEL
LIN {X 0,Y 393.101,Z 685.03,A -85,B 0,C 180,E1 10472.5,E2 10472.5} C_VEL
LIN {X 0,Y 393.09,Z 685.03,A -85,B 0,C 180,E1 10479.847,E2 10479.847} C_VEL
LIN {X 0,Y 392.985,Z 685.03,A -85,B 0,C 180,E1 10486.839,E2 10486.839} C_VEL
LIN {X 0,Y 393.009,Z 685.03,A -85,B 0,C 180,E1 10488.385,E2 10488.385} C_VEL
LIN {X 0,Y 395.402,Z 690.678,A -85,B 0,C 180,E1 10489.024,E2 10489.024} C_VEL
LIN {X 0,Y 410.394,Z 723.133,A -85,B 0,C 180,E1 10493.165,E2 10493.165} C_VEL
LIN {X 0,Y 420.173,Z 752.149,A -85,B 0,C 180,E1 10497,E2 10497} C_VEL
LIN {X 0,Y 414.569,Z 783.013,A -85,B 0,C 180,E1 10500.193,E2 10500.193} C_VEL
LIN {X 0,Y 408.617,Z 810.15,A -85,B 0,C 180,E1 10504.077,E2 10504.077} C_VEL
LIN {X 0,Y 403.373,Z 832.617,A -85,B 0,C 180,E1 10508.537,E2 10508.537} C_VEL
LIN {X 0,Y 399.456,Z 850.271,A -85,B 0,C 180,E1 10513.541,E2 10513.541} C_VEL
LIN {X 0,Y 397.053,Z 863.128,A -85,B 0,C 180,E1 10519.046,E2 10519.046} C_VEL
LIN {X 0,Y 396.049,Z 869.369,A -85,B 0,C 180,E1 10523.437,E2 10523.437} C_VEL
LIN {X 0,Y 395.79,Z 872.35,A -85,B 0,C 180,E1 10527.815,E2 10527.815} C_VEL
LIN {X 0,Y 395.824,Z 872.305,A -85,B 0,C 180,E1 10532.185,E2 10532.185} C_VEL
LIN {X 0,Y 396.339,Z 867.306,A -85,B 0,C 180,E1 10538.207,E2 10538.207} C_VEL
LIN {X 0,Y 397.973,Z 857.455,A -85,B 0,C 180,E1 10543.646,E2 10543.646} C_VEL
LIN {X 0,Y 400.977,Z 843.001,A -85,B 0,C 180,E1 10548.656,E2 10548.656} C_VEL
LIN {X 0,Y 405.767,Z 822.428,A -85,B 0,C 180,E1 10553.564,E2 10553.564} C_VEL
LIN {X 0,Y 411.138,Z 798.853,A -85,B 0,C 180,E1 10557.605,E2 10557.605} C_VEL
LIN {X 0,Y 417.244,Z 769.475,A -85,B 0,C 180,E1 10561.245,E2 10561.245} C_VEL
LIN {X 0,Y 419.992,Z 751.492,A -85,B 0,C 180,E1 10562.996,E2 10562.996} C_VEL
LIN {X 0,Y 409.895,Z 721.825,A -85,B 0,C 180,E1 10566.902,E2 10566.902} C_VEL
LIN {X 0,Y 395.172,Z 690.327,A -85,B 0,C 180,E1 10570.922,E2 10570.922} C_VEL
LIN {X 0,Y 393.039,Z 685.03,A -85,B 0,C 180,E1 10571.606,E2 10571.606} C_VEL
LIN {X 0,Y 393.042,Z 685.03,A -85,B 0,C 180,E1 10576.841,E2 10576.841} C_VEL
LIN {X 0,Y 393.056,Z 685.03,A -85,B 0,C 180,E1 10583.728,E2 10583.728} C_VEL
LIN {X 0,Y 393.175,Z 685.03,A -85,B 0,C 180,E1 10590.078,E2 10590.078} C_VEL
LIN {X 0,Y 393.432,Z 685.03,A -85,B 0,C 180,E1 10597.453,E2 10597.453} C_VEL
LIN {X 0,Y 393.81,Z 685.03,A -85,B 0,C 180,E1 10604.447,E2 10604.447} C_VEL
LIN {X 0,Y 393.999,Z 685.03,A -85,B 0,C 180,E1 10611.193,E2 10611.193} C_VEL
LIN {X 0,Y 394.264,Z 685.03,A -85,B 0,C 180,E1 10617.811,E2 10617.811} C_VEL
